(* Logix 5000 project; controller reports 1756-L63 rev 20.11; software revision 20.04; part 49 of 52 *)

        [172].log_data[23].time := 3600.0, [172].log_data[23].valid := 1, [172].log_data[24].time := 3600.0, [172].log_data[24].valid := 1, [172].log_data[25].time := 3600.0, [172].log_data[25].valid := 1, [172].log_data[26].time := 3600.0, [172].log_data[26].valid := 1, [172].log_data[27].time := 3600.0, [172].log_data[27].valid := 1, [172].log_data[28].time := 3600.0, [172].log_data[28].valid := 1, [172].log_data[29].min := 1.0, [172].log_data[29].max := 1.0, [172].log_data[29].total := 3600.0, [172].log_data[29].time := 3600.0, [172].log_data[29].valid := 1, [172].log_data[30].min := 1.0, [172].log_data[30].max := 1.0, [172].log_data[30].total := 3600.0, [172].log_data[30].time := 3600.0, [172].log_data[30].valid := 1, [172].log_data[31].max := 1.0, [172].log_data[31].total := 1629.7471, [172].log_data[31].time := 3600.0, [172].log_data[31].maxminute := 1, [172].log_data[31].valid := 1, [172].log_data[32].max := 1.0, [172].log_data[32].total := 1452.2471, [172].log_data[32].time := 3600.0, [172].log_data[32].maxminute := 11, [172].log_data[32].valid := 1, [172].log_data[33].time := 3600.0, [172].log_data[33].valid := 1, [172].log_data[34].time := 3600.0, [172].log_data[34].valid := 1, [172].log_data[35].max := 1.0, [172].log_data[35].total := 1440.5, [172].log_data[35].time := 3600.0, [172].log_data[35].minminute := 2, [172].log_data[35].valid := 1, [172].log_data[36].max := 1.0, [172].log_data[36].total := 1629.7471, [172].log_data[36].time := 3600.0, [172].log_data[36].maxminute := 4, [172].log_data[36].valid := 1, [172].log_data[37].max := 6.994973, [172].log_data[37].total := 3548.4736, [172].log_data[37].time := 3600.0, [172].log_data[37].maxminute := 52, [172].log_data[37].valid := 1, [172].log_data[38].time := 3600.0, [172].log_data[38].valid := 1, [172].log_data[39].min := 0.9945885, [172].log_data[39].max := 1.0214411, [172].log_data[39].total := 3605.796, [172].log_data[39].time := 3600.0, [172].log_data[39].minminute := 44, [172].log_data[39].maxminute := 58, [172].log_data[39].valid := 1,
        [172].log_data[40].min := 7.5503016, [172].log_data[40].max := 7.5794306, [172].log_data[40].total := 27251.781, [172].log_data[40].time := 3600.0, [172].log_data[40].minminute := 51, [172].log_data[40].maxminute := 15, [172].log_data[40].valid := 1, [172].log_data[41].min := 0.07907203, [172].log_data[41].max := 0.10674902, [172].log_data[41].total := 334.01642, [172].log_data[41].time := 3600.0, [172].log_data[41].minminute := 58, [172].log_data[41].valid := 1, [172].log_data[42].min := 2.293056, [172].log_data[42].max := 2.2978847, [172].log_data[42].total := 8264.451, [172].log_data[42].time := 3600.0, [172].log_data[42].minminute := 29, [172].log_data[42].maxminute := 2, [172].log_data[42].valid := 1, [172].log_data[43].min := -0.27999878, [172].log_data[43].max := -0.26000214, [172].log_data[43].total := -954.9988, [172].log_data[43].time := 3600.0, [172].log_data[43].valid := 1, [172].log_data[44].min := -0.30000305, [172].log_data[44].max := -0.27999878, [172].log_data[44].total := -1079.6469, [172].log_data[44].time := 3600.0, [172].log_data[44].maxminute := 4, [172].log_data[44].valid := 1, [172].log_data[45].time := 3600.0, [172].log_data[45].valid := 1, [172].log_data[46].time := 3600.0, [172].log_data[46].valid := 1, [172].log_data[47].time := 3600.0, [172].log_data[47].valid := 1, [172].log_data[48].min := 6.583802, [172].log_data[48].max := 6.9311595, [172].log_data[48].total := 24306.4, [172].log_data[48].time := 3600.0, [172].log_data[48].minminute := 5, [172].log_data[48].maxminute := 59, [172].log_data[48].valid := 1, [172].log_data[49].min := 6.690951, [172].log_data[49].max := 9.500274, [172].log_data[49].total := 31090.45, [172].log_data[49].time := 3600.0, [172].log_data[49].maxminute := 53, [172].log_data[49].valid := 1, [172].log_data[50].min := 2.067046, [172].log_data[50].max := 2.172219, [172].log_data[50].total := 7593.68, [172].log_data[50].time := 3600.0, [172].log_data[50].minminute := 51, [172].log_data[50].maxminute := 59, [172].log_data[50].valid := 1, [172].log_data[51].time := 3600.0, [172].log_data[51].valid := 1, [172].log_data[52].min := -3.0,
        [172].log_data[52].max := 0.11999512, [172].log_data[52].total := -7550.291, [172].log_data[52].time := 3600.0, [172].log_data[52].minminute := 43, [172].log_data[52].valid := 1, [172].log_data[53].min := -2.5, [172].log_data[53].max := 0.2599945, [172].log_data[53].total := -7057.6147, [172].log_data[53].time := 3600.0, [172].log_data[53].minminute := 14, [172].log_data[53].maxminute := 35, [172].log_data[53].valid := 1, [172].log_data[54].max := 0.56, [172].log_data[54].total := 1221.5302, [172].log_data[54].time := 3600.0, [172].log_data[54].maxminute := 1, [172].log_data[54].valid := 1, [172].log_data[55].max := 0.55799997, [172].log_data[55].total := 1217.0685, [172].log_data[55].time := 3600.0, [172].log_data[55].minminute := 2, [172].log_data[55].maxminute := 14, [172].log_data[55].valid := 1, [172].log_data[56].min := 0.16067745, [172].log_data[56].max := 0.16114853, [172].log_data[56].total := 579.2485, [172].log_data[56].time := 3600.0, [172].log_data[56].minminute := 9, [172].log_data[56].maxminute := 1, [172].log_data[56].valid := 1, [172].log_data[57].min := 0.34574097, [172].log_data[57].max := 0.3479787, [172].log_data[57].total := 1245.9099, [172].log_data[57].time := 3600.0, [172].log_data[57].minminute := 14, [172].log_data[57].maxminute := 1, [172].log_data[57].valid := 1, [172].log_data[58].time := 3600.0, [172].log_data[58].valid := 1, [172].log_data[59].time := 3600.0, [172].log_data[59].valid := 1, [172].log_data[60].valid := 1, [172].log_data[61].valid := 1, [172].log_data[62].valid := 1, [172].log_data[63].valid := 1, [172].log_data[64].valid := 1, [172].log_data[65].valid := 1, [172].log_data[66].valid := 1, [172].log_data[67].valid := 1, [172].log_data[68].valid := 1, [172].log_data[69].valid := 1, [172].log_data[70].valid := 1, [172].log_data[71].valid := 1, [172].log_data[72].valid := 1, [172].log_data[73].valid := 1, [172].log_data[74].valid := 1, [172].log_data[75].valid := 1, [172].log_data[76].valid := 1, [172].log_data[77].valid := 1, [172].log_data[78].valid := 1,
        [172].log_data[79].valid := 1, [172].log_data[80].valid := 1, [172].log_data[81].valid := 1, [172].log_data[82].valid := 1, [172].log_data[83].valid := 1, [172].log_data[84].valid := 1, [172].log_data[85].valid := 1, [172].log_data[86].valid := 1, [172].log_data[87].valid := 1, [172].log_data[88].valid := 1, [172].log_data[89].valid := 1, [172].log_data[90].valid := 1, [172].log_data[91].valid := 1, [172].log_data[92].valid := 1, [172].log_data[93].valid := 1, [172].log_data[94].valid := 1, [172].log_data[95].valid := 1, [172].log_data[96].valid := 1, [172].log_data[97].valid := 1, [172].log_data[98].valid := 1, [172].log_data[99].valid := 1, [172].log_data[100].valid := 1, [172].log_data[101].valid := 1, [172].log_data[102].valid := 1, [172].log_data[103].valid := 1, [172].log_data[104].valid := 1, [172].log_data[105].valid := 1, [172].log_data[106].valid := 1, [172].log_data[107].valid := 1, [172].log_data[108].valid := 1, [172].log_data[109].valid := 1, [172].log_data[110].valid := 1, [172].log_data[111].valid := 1, [172].log_data[112].valid := 1, [172].log_data[113].valid := 1, [172].log_data[114].valid := 1, [172].log_data[115].valid := 1, [172].log_data[116].valid := 1, [172].log_data[117].valid := 1, [172].log_data[118].valid := 1, [172].log_data[119].valid := 1, [172].log_data[120].valid := 1, [172].log_data[121].valid := 1, [172].log_data[122].valid := 1, [172].log_data[123].valid := 1, [172].log_data[124].valid := 1, [172].time.Year := 2023, [172].time.Month := 1, [172].time.Day := 11, [172].time.Hour := 23, [172].time.Minute := 59, [172].time.Second := 59, [173].log_data[0].min := 1.0, [173].log_data[0].max := 1.0, [173].log_data[0].total := 3600.0, [173].log_data[0].time := 3600.0, [173].log_data[0].valid := 1, [173].log_data[1].max := 1.0, [173].log_data[1].total := 26.251, [173].log_data[1].time := 3600.0,
        [173].log_data[1].valid := 1, [173].log_data[2].max := 1.0, [173].log_data[2].total := 26.251, [173].log_data[2].time := 3600.0, [173].log_data[2].valid := 1, [173].log_data[3].time := 3600.0, [173].log_data[3].valid := 1, [173].log_data[4].time := 3600.0, [173].log_data[4].valid := 1, [173].log_data[5].time := 3600.0, [173].log_data[5].valid := 1, [173].log_data[6].time := 3600.0, [173].log_data[6].valid := 1, [173].log_data[7].time := 3600.0, [173].log_data[7].valid := 1, [173].log_data[8].min := 1.0, [173].log_data[8].max := 1.0, [173].log_data[8].total := 3600.0, [173].log_data[8].time := 3600.0, [173].log_data[8].valid := 1, [173].log_data[9].min := 1.0, [173].log_data[9].max := 1.0, [173].log_data[9].total := 3600.0, [173].log_data[9].time := 3600.0, [173].log_data[9].valid := 1, [173].log_data[10].min := 1.0, [173].log_data[10].max := 1.0, [173].log_data[10].total := 3600.0, [173].log_data[10].time := 3600.0, [173].log_data[10].valid := 1, [173].log_data[11].time := 3600.0, [173].log_data[11].valid := 1, [173].log_data[12].min := 1.0, [173].log_data[12].max := 1.0, [173].log_data[12].total := 3600.0, [173].log_data[12].time := 3600.0, [173].log_data[12].valid := 1, [173].log_data[13].min := 1.0, [173].log_data[13].max := 1.0, [173].log_data[13].total := 3600.0, [173].log_data[13].time := 3600.0, [173].log_data[13].valid := 1, [173].log_data[14].time := 3600.0, [173].log_data[14].valid := 1, [173].log_data[15].time := 3600.0, [173].log_data[15].valid := 1, [173].log_data[16].time := 3600.0, [173].log_data[16].valid := 1, [173].log_data[17].min := 1.0, [173].log_data[17].max := 1.0, [173].log_data[17].total := 3600.0, [173].log_data[17].time := 3600.0, [173].log_data[17].valid := 1, [173].log_data[18].time := 3600.0, [173].log_data[18].valid := 1, [173].log_data[19].time := 3600.0, [173].log_data[19].valid := 1, [173].log_data[20].time := 3600.0, [173].log_data[20].valid := 1, [173].log_data[21].min := 1.0,
        [173].log_data[21].max := 1.0, [173].log_data[21].total := 3600.0, [173].log_data[21].time := 3600.0, [173].log_data[21].valid := 1, [173].log_data[22].time := 3600.0, [173].log_data[22].valid := 1, [173].log_data[23].time := 3600.0, [173].log_data[23].valid := 1, [173].log_data[24].time := 3600.0, [173].log_data[24].valid := 1, [173].log_data[25].time := 3600.0, [173].log_data[25].valid := 1, [173].log_data[26].time := 3600.0, [173].log_data[26].valid := 1, [173].log_data[27].time := 3600.0, [173].log_data[27].valid := 1, [173].log_data[28].time := 3600.0, [173].log_data[28].valid := 1, [173].log_data[29].min := 1.0, [173].log_data[29].max := 1.0, [173].log_data[29].total := 3600.0, [173].log_data[29].time := 3600.0, [173].log_data[29].valid := 1, [173].log_data[30].min := 1.0, [173].log_data[30].max := 1.0, [173].log_data[30].total := 3600.0, [173].log_data[30].time := 3600.0, [173].log_data[30].valid := 1, [173].log_data[31].max := 1.0, [173].log_data[31].total := 1629.7471, [173].log_data[31].time := 3600.0, [173].log_data[31].maxminute := 4, [173].log_data[31].valid := 1, [173].log_data[32].max := 1.0, [173].log_data[32].total := 1440.7471, [173].log_data[32].time := 3600.0, [173].log_data[32].minminute := 2, [173].log_data[32].valid := 1, [173].log_data[33].time := 3600.0, [173].log_data[33].valid := 1, [173].log_data[34].time := 3600.0, [173].log_data[34].valid := 1, [173].log_data[35].max := 1.0, [173].log_data[35].total := 1443.498, [173].log_data[35].time := 3600.0, [173].log_data[35].minminute := 5, [173].log_data[35].valid := 1, [173].log_data[36].max := 1.0, [173].log_data[36].total := 1629.7471, [173].log_data[36].time := 3600.0, [173].log_data[36].maxminute := 7, [173].log_data[36].valid := 1, [173].log_data[37].time := 3600.0, [173].log_data[37].valid := 1, [173].log_data[38].time := 3600.0, [173].log_data[38].valid := 1, [173].log_data[39].min := 0.995884, [173].log_data[39].max := 1.0066015, [173].log_data[39].total := 3607.993, [173].log_data[39].time := 3600.0,
        [173].log_data[39].minminute := 43, [173].log_data[39].maxminute := 56, [173].log_data[39].valid := 1, [173].log_data[40].min := 7.553049, [173].log_data[40].max := 7.5832787, [173].log_data[40].total := 27256.387, [173].log_data[40].time := 3600.0, [173].log_data[40].minminute := 13, [173].log_data[40].maxminute := 18, [173].log_data[40].valid := 1, [173].log_data[41].min := 0.08005347, [173].log_data[41].max := 0.13226709, [173].log_data[41].total := 406.6626, [173].log_data[41].time := 3600.0, [173].log_data[41].maxminute := 31, [173].log_data[41].valid := 1, [173].log_data[42].min := 2.293056, [173].log_data[42].max := 2.2978847, [173].log_data[42].total := 8264.515, [173].log_data[42].time := 3600.0, [173].log_data[42].minminute := 12, [173].log_data[42].maxminute := 45, [173].log_data[42].valid := 1, [173].log_data[43].min := -0.27999878, [173].log_data[43].max := -0.26000214, [173].log_data[43].total := -953.048, [173].log_data[43].time := 3600.0, [173].log_data[43].valid := 1, [173].log_data[44].min := -0.30000305, [173].log_data[44].max := -0.27999878, [173].log_data[44].total := -1078.877, [173].log_data[44].time := 3600.0, [173].log_data[44].maxminute := 4, [173].log_data[44].valid := 1, [173].log_data[45].time := 3600.0, [173].log_data[45].valid := 1, [173].log_data[46].time := 3600.0, [173].log_data[46].valid := 1, [173].log_data[47].time := 3600.0, [173].log_data[47].valid := 1, [173].log_data[48].min := 6.5983667, [173].log_data[48].max := 6.903678, [173].log_data[48].total := 24199.447, [173].log_data[48].time := 3600.0, [173].log_data[48].minminute := 23, [173].log_data[48].valid := 1, [173].log_data[49].min := 6.840722, [173].log_data[49].max := 9.401342, [173].log_data[49].total := 29274.203, [173].log_data[49].time := 3600.0, [173].log_data[49].minminute := 20, [173].log_data[49].maxminute := 59, [173].log_data[49].valid := 1, [173].log_data[50].min := 2.0936632, [173].log_data[50].max := 2.1728077, [173].log_data[50].total := 7691.275, [173].log_data[50].time := 3600.0, [173].log_data[50].minminute := 59, [173].log_data[50].valid := 1, [173].log_data[51].time := 3600.0,
        [173].log_data[51].valid := 1, [173].log_data[52].min := -2.959999, [173].log_data[52].max := 0.11999512, [173].log_data[52].total := -7556.767, [173].log_data[52].time := 3600.0, [173].log_data[52].minminute := 25, [173].log_data[52].maxminute := 3, [173].log_data[52].valid := 1, [173].log_data[53].min := -2.5, [173].log_data[53].max := 0.2400055, [173].log_data[53].total := -7110.352, [173].log_data[53].time := 3600.0, [173].log_data[53].minminute := 42, [173].log_data[53].maxminute := 17, [173].log_data[53].valid := 1, [173].log_data[54].max := 0.528, [173].log_data[54].total := 1217.4906, [173].log_data[54].time := 3600.0, [173].log_data[54].minminute := 2, [173].log_data[54].maxminute := 25, [173].log_data[54].valid := 1, [173].log_data[55].max := 0.525, [173].log_data[55].total := 1220.6111, [173].log_data[55].time := 3600.0, [173].log_data[55].minminute := 5, [173].log_data[55].maxminute := 39, [173].log_data[55].valid := 1, [173].log_data[56].min := 0.1607167, [173].log_data[56].max := 0.16110928, [173].log_data[56].total := 579.1586, [173].log_data[56].time := 3600.0, [173].log_data[56].minminute := 47, [173].log_data[56].maxminute := 6, [173].log_data[56].valid := 1, [173].log_data[57].min := 0.3444062, [173].log_data[57].max := 0.34609428, [173].log_data[57].total := 1242.74, [173].log_data[57].time := 3600.0, [173].log_data[57].minminute := 35, [173].log_data[57].maxminute := 1, [173].log_data[57].valid := 1, [173].log_data[58].time := 3600.0, [173].log_data[58].valid := 1, [173].log_data[59].time := 3600.0, [173].log_data[59].valid := 1, [173].log_data[60].valid := 1, [173].log_data[61].valid := 1, [173].log_data[62].valid := 1, [173].log_data[63].valid := 1, [173].log_data[64].valid := 1, [173].log_data[65].valid := 1, [173].log_data[66].valid := 1, [173].log_data[67].valid := 1, [173].log_data[68].valid := 1, [173].log_data[69].valid := 1, [173].log_data[70].valid := 1, [173].log_data[71].valid := 1, [173].log_data[72].valid := 1, [173].log_data[73].valid := 1, [173].log_data[74].valid := 1,
        [173].log_data[75].valid := 1, [173].log_data[76].valid := 1, [173].log_data[77].valid := 1, [173].log_data[78].valid := 1, [173].log_data[79].valid := 1, [173].log_data[80].valid := 1, [173].log_data[81].valid := 1, [173].log_data[82].valid := 1, [173].log_data[83].valid := 1, [173].log_data[84].valid := 1, [173].log_data[85].valid := 1, [173].log_data[86].valid := 1, [173].log_data[87].valid := 1, [173].log_data[88].valid := 1, [173].log_data[89].valid := 1, [173].log_data[90].valid := 1, [173].log_data[91].valid := 1, [173].log_data[92].valid := 1, [173].log_data[93].valid := 1, [173].log_data[94].valid := 1, [173].log_data[95].valid := 1, [173].log_data[96].valid := 1, [173].log_data[97].valid := 1, [173].log_data[98].valid := 1, [173].log_data[99].valid := 1, [173].log_data[100].valid := 1, [173].log_data[101].valid := 1, [173].log_data[102].valid := 1, [173].log_data[103].valid := 1, [173].log_data[104].valid := 1, [173].log_data[105].valid := 1, [173].log_data[106].valid := 1, [173].log_data[107].valid := 1, [173].log_data[108].valid := 1, [173].log_data[109].valid := 1, [173].log_data[110].valid := 1, [173].log_data[111].valid := 1, [173].log_data[112].valid := 1, [173].log_data[113].valid := 1, [173].log_data[114].valid := 1, [173].log_data[115].valid := 1, [173].log_data[116].valid := 1, [173].log_data[117].valid := 1, [173].log_data[118].valid := 1, [173].log_data[119].valid := 1, [173].log_data[120].valid := 1, [173].log_data[121].valid := 1, [173].log_data[122].valid := 1, [173].log_data[123].valid := 1, [173].log_data[124].valid := 1, [173].time.Year := 2023, [173].time.Month := 1, [173].time.Day := 12, [173].time.Minute := 59, [173].time.Second := 59, [174].log_data[0].min := 1.0, [174].log_data[0].max := 1.0, [174].log_data[0].total := 3599.5, [174].log_data[0].time := 3599.5, [174].log_data[0].valid := 1,
        [174].log_data[1].time := 3599.5, [174].log_data[1].valid := 1, [174].log_data[2].time := 3599.5, [174].log_data[2].valid := 1, [174].log_data[3].time := 3599.5, [174].log_data[3].valid := 1, [174].log_data[4].time := 3599.5, [174].log_data[4].valid := 1, [174].log_data[5].time := 3599.5, [174].log_data[5].valid := 1, [174].log_data[6].time := 3599.5, [174].log_data[6].valid := 1, [174].log_data[7].time := 3599.5, [174].log_data[7].valid := 1, [174].log_data[8].min := 1.0, [174].log_data[8].max := 1.0, [174].log_data[8].total := 3599.5, [174].log_data[8].time := 3599.5, [174].log_data[8].valid := 1, [174].log_data[9].min := 1.0, [174].log_data[9].max := 1.0, [174].log_data[9].total := 3599.5, [174].log_data[9].time := 3599.5, [174].log_data[9].valid := 1, [174].log_data[10].min := 1.0, [174].log_data[10].max := 1.0, [174].log_data[10].total := 3599.5, [174].log_data[10].time := 3599.5, [174].log_data[10].valid := 1, [174].log_data[11].time := 3599.5, [174].log_data[11].valid := 1, [174].log_data[12].min := 1.0, [174].log_data[12].max := 1.0, [174].log_data[12].total := 3599.5, [174].log_data[12].time := 3599.5, [174].log_data[12].valid := 1, [174].log_data[13].min := 1.0, [174].log_data[13].max := 1.0, [174].log_data[13].total := 3599.5, [174].log_data[13].time := 3599.5, [174].log_data[13].valid := 1, [174].log_data[14].time := 3599.5, [174].log_data[14].valid := 1, [174].log_data[15].time := 3599.5, [174].log_data[15].valid := 1, [174].log_data[16].time := 3599.5, [174].log_data[16].valid := 1, [174].log_data[17].min := 1.0, [174].log_data[17].max := 1.0, [174].log_data[17].total := 3599.5, [174].log_data[17].time := 3599.5, [174].log_data[17].valid := 1, [174].log_data[18].time := 3599.5, [174].log_data[18].valid := 1, [174].log_data[19].time := 3599.5, [174].log_data[19].valid := 1, [174].log_data[20].time := 3599.5, [174].log_data[20].valid := 1, [174].log_data[21].min := 1.0, [174].log_data[21].max := 1.0,
        [174].log_data[21].total := 3599.5, [174].log_data[21].time := 3599.5, [174].log_data[21].valid := 1, [174].log_data[22].time := 3599.5, [174].log_data[22].valid := 1, [174].log_data[23].time := 3599.5, [174].log_data[23].valid := 1, [174].log_data[24].time := 3599.5, [174].log_data[24].valid := 1, [174].log_data[25].time := 3599.5, [174].log_data[25].valid := 1, [174].log_data[26].time := 3599.5, [174].log_data[26].valid := 1, [174].log_data[27].time := 3599.5, [174].log_data[27].valid := 1, [174].log_data[28].time := 3599.5, [174].log_data[28].valid := 1, [174].log_data[29].min := 1.0, [174].log_data[29].max := 1.0, [174].log_data[29].total := 3599.5, [174].log_data[29].time := 3599.5, [174].log_data[29].valid := 1, [174].log_data[30].min := 1.0, [174].log_data[30].max := 1.0, [174].log_data[30].total := 3599.5, [174].log_data[30].time := 3599.5, [174].log_data[30].valid := 1, [174].log_data[31].max := 1.0, [174].log_data[31].total := 1629.7471, [174].log_data[31].time := 3599.5, [174].log_data[31].maxminute := 7, [174].log_data[31].valid := 1, [174].log_data[32].max := 1.0, [174].log_data[32].total := 1452.998, [174].log_data[32].time := 3599.5, [174].log_data[32].minminute := 6, [174].log_data[32].valid := 1, [174].log_data[33].time := 3599.5, [174].log_data[33].valid := 1, [174].log_data[34].time := 3599.5, [174].log_data[34].valid := 1, [174].log_data[35].max := 1.0, [174].log_data[35].total := 1629.7471, [174].log_data[35].time := 3599.5, [174].log_data[35].valid := 1, [174].log_data[36].max := 1.0, [174].log_data[36].total := 1525.7471, [174].log_data[36].time := 3599.5, [174].log_data[36].maxminute := 10, [174].log_data[36].valid := 1, [174].log_data[37].time := 3599.5, [174].log_data[37].valid := 1, [174].log_data[38].time := 3599.5, [174].log_data[38].valid := 1, [174].log_data[39].min := 0.9956484, [174].log_data[39].max := 1.0071905, [174].log_data[39].total := 3608.351, [174].log_data[39].time := 3599.5, [174].log_data[39].minminute := 10, [174].log_data[39].maxminute := 23,
        [174].log_data[39].valid := 1, [174].log_data[40].min := 7.5390344, [174].log_data[40].max := 7.592072, [174].log_data[40].total := 27246.436, [174].log_data[40].time := 3599.5, [174].log_data[40].minminute := 9, [174].log_data[40].maxminute := 18, [174].log_data[40].valid := 1, [174].log_data[41].min := 0.08613843, [174].log_data[41].max := 0.14345556, [174].log_data[41].total := 424.99884, [174].log_data[41].time := 3599.5, [174].log_data[41].minminute := 29, [174].log_data[41].maxminute := 56, [174].log_data[41].valid := 1, [174].log_data[42].min := 2.293056, [174].log_data[42].max := 2.2980025, [174].log_data[42].total := 8263.423, [174].log_data[42].time := 3599.5, [174].log_data[42].minminute := 20, [174].log_data[42].maxminute := 44, [174].log_data[42].valid := 1, [174].log_data[43].min := -0.27999878, [174].log_data[43].max := -0.26000214, [174].log_data[43].total := -944.1006, [174].log_data[43].time := 3599.5, [174].log_data[43].valid := 1, [174].log_data[44].min := -0.30000305, [174].log_data[44].max := -0.27999878, [174].log_data[44].total := -1079.4894, [174].log_data[44].time := 3599.5, [174].log_data[44].maxminute := 6, [174].log_data[44].valid := 1, [174].log_data[45].time := 3599.5, [174].log_data[45].valid := 1, [174].log_data[46].time := 3599.5, [174].log_data[46].valid := 1, [174].log_data[47].time := 3599.5, [174].log_data[47].valid := 1, [174].log_data[48].min := 6.753908, [174].log_data[48].max := 6.762702, [174].log_data[48].total := 24325.047, [174].log_data[48].time := 3599.5, [174].log_data[48].minminute := 58, [174].log_data[48].maxminute := 2, [174].log_data[48].valid := 1, [174].log_data[49].min := 9.398202, [174].log_data[49].max := 9.565442, [174].log_data[49].total := 34182.1, [174].log_data[49].time := 3599.5, [174].log_data[49].maxminute := 52, [174].log_data[49].valid := 1, [174].log_data[50].min := 2.006392, [174].log_data[50].max := 2.1013186, [174].log_data[50].total := 7397.241, [174].log_data[50].time := 3599.5, [174].log_data[50].minminute := 59, [174].log_data[50].valid := 1, [174].log_data[51].time := 3599.5, [174].log_data[51].valid := 1,
        [174].log_data[52].min := -3.0800018, [174].log_data[52].max := 0.11999512, [174].log_data[52].total := -7629.0737, [174].log_data[52].time := 3599.5, [174].log_data[52].minminute := 7, [174].log_data[52].maxminute := 6, [174].log_data[52].valid := 1, [174].log_data[53].min := -2.5200043, [174].log_data[53].max := 0.19999695, [174].log_data[53].total := -7349.1704, [174].log_data[53].time := 3599.5, [174].log_data[53].minminute := 57, [174].log_data[53].valid := 1, [174].log_data[54].max := 0.559, [174].log_data[54].total := 1224.2659, [174].log_data[54].time := 3599.5, [174].log_data[54].minminute := 6, [174].log_data[54].maxminute := 7, [174].log_data[54].valid := 1, [174].log_data[55].max := 0.528, [174].log_data[55].total := 1250.9253, [174].log_data[55].time := 3599.5, [174].log_data[55].maxminute := 31, [174].log_data[55].valid := 1, [174].log_data[56].min := 0.16067745, [174].log_data[56].max := 0.16110928, [174].log_data[56].total := 578.99304, [174].log_data[56].time := 3599.5, [174].log_data[56].minminute := 34, [174].log_data[56].maxminute := 6, [174].log_data[56].valid := 1, [174].log_data[57].min := 0.3444062, [174].log_data[57].max := 0.34483802, [174].log_data[57].total := 1240.3518, [174].log_data[57].time := 3599.5, [174].log_data[57].minminute := 38, [174].log_data[57].maxminute := 11, [174].log_data[57].valid := 1, [174].log_data[58].time := 3599.5, [174].log_data[58].valid := 1, [174].log_data[59].time := 3599.5, [174].log_data[59].valid := 1, [174].log_data[60].valid := 1, [174].log_data[61].valid := 1, [174].log_data[62].valid := 1, [174].log_data[63].valid := 1, [174].log_data[64].valid := 1, [174].log_data[65].valid := 1, [174].log_data[66].valid := 1, [174].log_data[67].valid := 1, [174].log_data[68].valid := 1, [174].log_data[69].valid := 1, [174].log_data[70].valid := 1, [174].log_data[71].valid := 1, [174].log_data[72].valid := 1, [174].log_data[73].valid := 1, [174].log_data[74].valid := 1, [174].log_data[75].valid := 1, [174].log_data[76].valid := 1, [174].log_data[77].valid := 1,
        [174].log_data[78].valid := 1, [174].log_data[79].valid := 1, [174].log_data[80].valid := 1, [174].log_data[81].valid := 1, [174].log_data[82].valid := 1, [174].log_data[83].valid := 1, [174].log_data[84].valid := 1, [174].log_data[85].valid := 1, [174].log_data[86].valid := 1, [174].log_data[87].valid := 1, [174].log_data[88].valid := 1, [174].log_data[89].valid := 1, [174].log_data[90].valid := 1, [174].log_data[91].valid := 1, [174].log_data[92].valid := 1, [174].log_data[93].valid := 1, [174].log_data[94].valid := 1, [174].log_data[95].valid := 1, [174].log_data[96].valid := 1, [174].log_data[97].valid := 1, [174].log_data[98].valid := 1, [174].log_data[99].valid := 1, [174].log_data[100].valid := 1, [174].log_data[101].valid := 1, [174].log_data[102].valid := 1, [174].log_data[103].valid := 1, [174].log_data[104].valid := 1, [174].log_data[105].valid := 1, [174].log_data[106].valid := 1, [174].log_data[107].valid := 1, [174].log_data[108].valid := 1, [174].log_data[109].valid := 1, [174].log_data[110].valid := 1, [174].log_data[111].valid := 1, [174].log_data[112].valid := 1, [174].log_data[113].valid := 1, [174].log_data[114].valid := 1, [174].log_data[115].valid := 1, [174].log_data[116].valid := 1, [174].log_data[117].valid := 1, [174].log_data[118].valid := 1, [174].log_data[119].valid := 1, [174].log_data[120].valid := 1, [174].log_data[121].valid := 1, [174].log_data[122].valid := 1, [174].log_data[123].valid := 1, [174].log_data[124].valid := 1, [174].time.Year := 2023, [174].time.Month := 1, [174].time.Day := 12, [174].time.Hour := 1, [174].time.Minute := 59, [174].time.Second := 59, [175].log_data[0].min := 1.0, [175].log_data[0].max := 1.0, [175].log_data[0].total := 3600.0, [175].log_data[0].time := 3600.0, [175].log_data[0].valid := 1, [175].log_data[1].max := 1.0, [175].log_data[1].total := 524.0,
        [175].log_data[1].time := 3600.0, [175].log_data[1].maxminute := 21, [175].log_data[1].valid := 1, [175].log_data[2].max := 1.0, [175].log_data[2].total := 520.5, [175].log_data[2].time := 3600.0, [175].log_data[2].maxminute := 21, [175].log_data[2].valid := 1, [175].log_data[3].time := 3600.0, [175].log_data[3].valid := 1, [175].log_data[4].time := 3600.0, [175].log_data[4].valid := 1, [175].log_data[5].max := 1.0, [175].log_data[5].total := 237.0, [175].log_data[5].time := 3600.0, [175].log_data[5].maxminute := 23, [175].log_data[5].valid := 1, [175].log_data[6].time := 3600.0, [175].log_data[6].valid := 1, [175].log_data[7].time := 3600.0, [175].log_data[7].valid := 1, [175].log_data[8].max := 1.0, [175].log_data[8].total := 2444.5, [175].log_data[8].time := 3600.0, [175].log_data[8].minminute := 5, [175].log_data[8].valid := 1, [175].log_data[9].max := 1.0, [175].log_data[9].total := 2441.0, [175].log_data[9].time := 3600.0, [175].log_data[9].minminute := 5, [175].log_data[9].valid := 1, [175].log_data[10].min := 1.0, [175].log_data[10].max := 1.0, [175].log_data[10].total := 3600.0, [175].log_data[10].time := 3600.0, [175].log_data[10].valid := 1, [175].log_data[11].time := 3600.0, [175].log_data[11].valid := 1, [175].log_data[12].min := 1.0, [175].log_data[12].max := 1.0, [175].log_data[12].total := 3600.0, [175].log_data[12].time := 3600.0, [175].log_data[12].valid := 1, [175].log_data[13].min := 1.0, [175].log_data[13].max := 1.0, [175].log_data[13].total := 3600.0, [175].log_data[13].time := 3600.0, [175].log_data[13].valid := 1, [175].log_data[14].time := 3600.0, [175].log_data[14].valid := 1, [175].log_data[15].time := 3600.0, [175].log_data[15].valid := 1, [175].log_data[16].time := 3600.0, [175].log_data[16].valid := 1, [175].log_data[17].min := 1.0, [175].log_data[17].max := 1.0, [175].log_data[17].total := 3600.0, [175].log_data[17].time := 3600.0, [175].log_data[17].valid := 1, [175].log_data[18].time := 3600.0,
        [175].log_data[18].valid := 1, [175].log_data[19].time := 3600.0, [175].log_data[19].valid := 1, [175].log_data[20].time := 3600.0, [175].log_data[20].valid := 1, [175].log_data[21].min := 1.0, [175].log_data[21].max := 1.0, [175].log_data[21].total := 3600.0, [175].log_data[21].time := 3600.0, [175].log_data[21].valid := 1, [175].log_data[22].time := 3600.0, [175].log_data[22].valid := 1, [175].log_data[23].time := 3600.0, [175].log_data[23].valid := 1, [175].log_data[24].time := 3600.0, [175].log_data[24].valid := 1, [175].log_data[25].time := 3600.0, [175].log_data[25].valid := 1, [175].log_data[26].time := 3600.0, [175].log_data[26].valid := 1, [175].log_data[27].time := 3600.0, [175].log_data[27].valid := 1, [175].log_data[28].time := 3600.0, [175].log_data[28].valid := 1, [175].log_data[29].min := 1.0, [175].log_data[29].max := 1.0, [175].log_data[29].total := 3600.0, [175].log_data[29].time := 3600.0, [175].log_data[29].valid := 1, [175].log_data[30].min := 1.0, [175].log_data[30].max := 1.0, [175].log_data[30].total := 3600.0, [175].log_data[30].time := 3600.0, [175].log_data[30].valid := 1, [175].log_data[31].max := 1.0, [175].log_data[31].total := 736.998, [175].log_data[31].time := 3600.0, [175].log_data[31].maxminute := 25, [175].log_data[31].valid := 1, [175].log_data[32].max := 1.0, [175].log_data[32].total := 1426.998, [175].log_data[32].time := 3600.0, [175].log_data[32].valid := 1, [175].log_data[33].time := 3600.0, [175].log_data[33].valid := 1, [175].log_data[34].time := 3600.0, [175].log_data[34].valid := 1, [175].log_data[35].max := 1.0, [175].log_data[35].total := 1064.247, [175].log_data[35].time := 3600.0, [175].log_data[35].maxminute := 3, [175].log_data[35].valid := 1, [175].log_data[36].max := 1.0, [175].log_data[36].total := 1020.498, [175].log_data[36].time := 3600.0, [175].log_data[36].minminute := 1, [175].log_data[36].valid := 1, [175].log_data[37].max := 7.558722, [175].log_data[37].total := 3407.4478, [175].log_data[37].time := 3600.0,
        [175].log_data[37].maxminute := 21, [175].log_data[37].valid := 1, [175].log_data[38].time := 3600.0, [175].log_data[38].valid := 1, [175].log_data[39].min := 0.9945885, [175].log_data[39].max := 1.02097, [175].log_data[39].total := 3608.6638, [175].log_data[39].time := 3600.0, [175].log_data[39].minminute := 51, [175].log_data[39].maxminute := 23, [175].log_data[39].valid := 1, [175].log_data[40].min := 7.5379353, [175].log_data[40].max := 7.5794306, [175].log_data[40].total := 27251.215, [175].log_data[40].time := 3600.0, [175].log_data[40].minminute := 14, [175].log_data[40].maxminute := 16, [175].log_data[40].valid := 1, [175].log_data[41].min := 0.0963457, [175].log_data[41].max := 0.14031494, [175].log_data[41].total := 379.17615, [175].log_data[41].time := 3600.0, [175].log_data[41].minminute := 52, [175].log_data[41].valid := 1, [175].log_data[42].min := 2.2929382, [175].log_data[42].max := 2.2978847, [175].log_data[42].total := 8264.402, [175].log_data[42].time := 3600.0, [175].log_data[42].minminute := 46, [175].log_data[42].maxminute := 4, [175].log_data[42].valid := 1, [175].log_data[43].min := -0.27999878, [175].log_data[43].max := -0.26000214, [175].log_data[43].total := -943.9623, [175].log_data[43].time := 3600.0, [175].log_data[43].valid := 1, [175].log_data[44].min := -0.30000305, [175].log_data[44].max := -0.27999878, [175].log_data[44].total := -1079.5896, [175].log_data[44].time := 3600.0, [175].log_data[44].valid := 1, [175].log_data[45].time := 3600.0, [175].log_data[45].valid := 1, [175].log_data[46].time := 3600.0, [175].log_data[46].valid := 1, [175].log_data[47].time := 3600.0, [175].log_data[47].valid := 1, [175].log_data[48].min := 6.5810537, [175].log_data[48].max := 6.969357, [175].log_data[48].total := 24223.447, [175].log_data[48].time := 3600.0, [175].log_data[48].minminute := 53, [175].log_data[48].maxminute := 26, [175].log_data[48].valid := 1, [175].log_data[49].min := 6.7979293, [175].log_data[49].max := 9.501255, [175].log_data[49].total := 30011.445, [175].log_data[49].time := 3600.0, [175].log_data[49].minminute := 49, [175].log_data[49].valid := 1,
        [175].log_data[50].min := 1.9999144, [175].log_data[50].max := 2.1501951, [175].log_data[50].total := 7513.3774, [175].log_data[50].time := 3600.0, [175].log_data[50].minminute := 5, [175].log_data[50].maxminute := 25, [175].log_data[50].valid := 1, [175].log_data[51].time := 3600.0, [175].log_data[51].valid := 1, [175].log_data[52].min := -4.1800003, [175].log_data[52].max := 0.11999512, [175].log_data[52].total := -6929.6797, [175].log_data[52].time := 3600.0, [175].log_data[52].minminute := 25, [175].log_data[52].valid := 1, [175].log_data[53].min := -3.9199982, [175].log_data[53].max := 0.19999695, [175].log_data[53].total := -6288.31, [175].log_data[53].time := 3600.0, [175].log_data[53].minminute := 25, [175].log_data[53].maxminute := 32, [175].log_data[53].valid := 1, [175].log_data[54].max := 0.51, [175].log_data[54].total := 855.8069, [175].log_data[54].time := 3600.0, [175].log_data[54].valid := 1, [175].log_data[55].max := 0.514, [175].log_data[55].total := 824.69495, [175].log_data[55].time := 3600.0, [175].log_data[55].minminute := 1, [175].log_data[55].maxminute := 33, [175].log_data[55].valid := 1, [175].log_data[56].min := 0.16063818, [175].log_data[56].max := 0.16107002, [175].log_data[56].total := 578.963, [175].log_data[56].time := 3600.0, [175].log_data[56].minminute := 56, [175].log_data[56].maxminute := 6, [175].log_data[56].valid := 1, [175].log_data[57].min := 0.3431499, [175].log_data[57].max := 0.34483802, [175].log_data[57].total := 1240.1224, [175].log_data[57].time := 3600.0, [175].log_data[57].minminute := 59, [175].log_data[57].maxminute := 43, [175].log_data[57].valid := 1, [175].log_data[58].time := 3600.0, [175].log_data[58].valid := 1, [175].log_data[59].time := 3600.0, [175].log_data[59].valid := 1, [175].log_data[60].valid := 1, [175].log_data[61].valid := 1, [175].log_data[62].valid := 1, [175].log_data[63].valid := 1, [175].log_data[64].valid := 1, [175].log_data[65].valid := 1, [175].log_data[66].valid := 1, [175].log_data[67].valid := 1, [175].log_data[68].valid := 1, [175].log_data[69].valid := 1,
        [175].log_data[70].valid := 1, [175].log_data[71].valid := 1, [175].log_data[72].valid := 1, [175].log_data[73].valid := 1, [175].log_data[74].valid := 1, [175].log_data[75].valid := 1, [175].log_data[76].valid := 1, [175].log_data[77].valid := 1, [175].log_data[78].valid := 1, [175].log_data[79].valid := 1, [175].log_data[80].valid := 1, [175].log_data[81].valid := 1, [175].log_data[82].valid := 1, [175].log_data[83].valid := 1, [175].log_data[84].valid := 1, [175].log_data[85].valid := 1, [175].log_data[86].valid := 1, [175].log_data[87].valid := 1, [175].log_data[88].valid := 1, [175].log_data[89].valid := 1, [175].log_data[90].valid := 1, [175].log_data[91].valid := 1, [175].log_data[92].valid := 1, [175].log_data[93].valid := 1, [175].log_data[94].valid := 1, [175].log_data[95].valid := 1, [175].log_data[96].valid := 1, [175].log_data[97].valid := 1, [175].log_data[98].valid := 1, [175].log_data[99].valid := 1, [175].log_data[100].valid := 1, [175].log_data[101].valid := 1, [175].log_data[102].valid := 1, [175].log_data[103].valid := 1, [175].log_data[104].valid := 1, [175].log_data[105].valid := 1, [175].log_data[106].valid := 1, [175].log_data[107].valid := 1, [175].log_data[108].valid := 1, [175].log_data[109].valid := 1, [175].log_data[110].valid := 1, [175].log_data[111].valid := 1, [175].log_data[112].valid := 1, [175].log_data[113].valid := 1, [175].log_data[114].valid := 1, [175].log_data[115].valid := 1, [175].log_data[116].valid := 1, [175].log_data[117].valid := 1, [175].log_data[118].valid := 1, [175].log_data[119].valid := 1, [175].log_data[120].valid := 1, [175].log_data[121].valid := 1, [175].log_data[122].valid := 1, [175].log_data[123].valid := 1, [175].log_data[124].valid := 1, [175].time.Year := 2023, [175].time.Month := 1, [175].time.Day := 12, [175].time.Hour := 2, [175].time.Minute := 59,
        [175].time.Second := 59, [176].log_data[0].min := 1.0, [176].log_data[0].max := 1.0, [176].log_data[0].total := 3600.0, [176].log_data[0].time := 3600.0, [176].log_data[0].valid := 1, [176].log_data[1].time := 3600.0, [176].log_data[1].valid := 1, [176].log_data[2].time := 3600.0, [176].log_data[2].valid := 1, [176].log_data[3].time := 3600.0, [176].log_data[3].valid := 1, [176].log_data[4].time := 3600.0, [176].log_data[4].valid := 1, [176].log_data[5].time := 3600.0, [176].log_data[5].valid := 1, [176].log_data[6].time := 3600.0, [176].log_data[6].valid := 1, [176].log_data[7].time := 3600.0, [176].log_data[7].valid := 1, [176].log_data[8].max := 1.0, [176].log_data[8].total := 2797.251, [176].log_data[8].time := 3600.0, [176].log_data[8].minminute := 46, [176].log_data[8].valid := 1, [176].log_data[9].max := 1.0, [176].log_data[9].total := 2797.251, [176].log_data[9].time := 3600.0, [176].log_data[9].minminute := 46, [176].log_data[9].valid := 1, [176].log_data[10].min := 1.0, [176].log_data[10].max := 1.0, [176].log_data[10].total := 3600.0, [176].log_data[10].time := 3600.0, [176].log_data[10].valid := 1, [176].log_data[11].time := 3600.0, [176].log_data[11].valid := 1, [176].log_data[12].min := 1.0, [176].log_data[12].max := 1.0, [176].log_data[12].total := 3600.0, [176].log_data[12].time := 3600.0, [176].log_data[12].valid := 1, [176].log_data[13].min := 1.0, [176].log_data[13].max := 1.0, [176].log_data[13].total := 3600.0, [176].log_data[13].time := 3600.0, [176].log_data[13].valid := 1, [176].log_data[14].time := 3600.0, [176].log_data[14].valid := 1, [176].log_data[15].time := 3600.0, [176].log_data[15].valid := 1, [176].log_data[16].time := 3600.0, [176].log_data[16].valid := 1, [176].log_data[17].min := 1.0, [176].log_data[17].max := 1.0, [176].log_data[17].total := 3600.0, [176].log_data[17].time := 3600.0, [176].log_data[17].valid := 1, [176].log_data[18].time := 3600.0, [176].log_data[18].valid := 1,
        [176].log_data[19].time := 3600.0, [176].log_data[19].valid := 1, [176].log_data[20].time := 3600.0, [176].log_data[20].valid := 1, [176].log_data[21].min := 1.0, [176].log_data[21].max := 1.0, [176].log_data[21].total := 3600.0, [176].log_data[21].time := 3600.0, [176].log_data[21].valid := 1, [176].log_data[22].time := 3600.0, [176].log_data[22].valid := 1, [176].log_data[23].time := 3600.0, [176].log_data[23].valid := 1, [176].log_data[24].time := 3600.0, [176].log_data[24].valid := 1, [176].log_data[25].time := 3600.0, [176].log_data[25].valid := 1, [176].log_data[26].time := 3600.0, [176].log_data[26].valid := 1, [176].log_data[27].time := 3600.0, [176].log_data[27].valid := 1, [176].log_data[28].time := 3600.0, [176].log_data[28].valid := 1, [176].log_data[29].min := 1.0, [176].log_data[29].max := 1.0, [176].log_data[29].total := 3600.0, [176].log_data[29].time := 3600.0, [176].log_data[29].valid := 1, [176].log_data[30].min := 1.0, [176].log_data[30].max := 1.0, [176].log_data[30].total := 3600.0, [176].log_data[30].time := 3600.0, [176].log_data[30].valid := 1, [176].log_data[31].max := 1.0, [176].log_data[31].total := 1263.749, [176].log_data[31].time := 3600.0, [176].log_data[31].maxminute := 1, [176].log_data[31].valid := 1, [176].log_data[32].max := 1.0, [176].log_data[32].total := 1095.749, [176].log_data[32].time := 3600.0, [176].log_data[32].valid := 1, [176].log_data[33].time := 3600.0, [176].log_data[33].valid := 1, [176].log_data[34].time := 3600.0, [176].log_data[34].valid := 1, [176].log_data[35].max := 1.0, [176].log_data[35].total := 1278.498, [176].log_data[35].time := 3600.0, [176].log_data[35].minminute := 3, [176].log_data[35].valid := 1, [176].log_data[36].max := 1.0, [176].log_data[36].total := 1086.498, [176].log_data[36].time := 3600.0, [176].log_data[36].maxminute := 4, [176].log_data[36].valid := 1, [176].log_data[37].time := 3600.0, [176].log_data[37].valid := 1, [176].log_data[38].time := 3600.0, [176].log_data[38].valid := 1,
        [176].log_data[39].min := 0.9941174, [176].log_data[39].max := 1.0041281, [176].log_data[39].total := 3599.7744, [176].log_data[39].time := 3600.0, [176].log_data[39].minminute := 27, [176].log_data[39].maxminute := 1, [176].log_data[39].valid := 1, [176].log_data[40].min := 7.5503016, [176].log_data[40].max := 7.5838275, [176].log_data[40].total := 27250.193, [176].log_data[40].time := 3600.0, [176].log_data[40].minminute := 30, [176].log_data[40].maxminute := 32, [176].log_data[40].valid := 1, [176].log_data[41].min := 0.09438281, [176].log_data[41].max := 0.12107837, [176].log_data[41].total := 379.78085, [176].log_data[41].time := 3600.0, [176].log_data[41].minminute := 1, [176].log_data[41].maxminute := 44, [176].log_data[41].valid := 1, [176].log_data[42].min := 2.2928205, [176].log_data[42].max := 2.2978847, [176].log_data[42].total := 8264.428, [176].log_data[42].time := 3600.0, [176].log_data[42].minminute := 54, [176].log_data[42].maxminute := 22, [176].log_data[42].valid := 1, [176].log_data[43].min := -0.27999878, [176].log_data[43].max := -0.26000214, [176].log_data[43].total := -969.35944, [176].log_data[43].time := 3600.0, [176].log_data[43].valid := 1, [176].log_data[44].min := -0.30000305, [176].log_data[44].max := -0.27999878, [176].log_data[44].total := -1080.0612, [176].log_data[44].time := 3600.0, [176].log_data[44].valid := 1, [176].log_data[45].time := 3600.0, [176].log_data[45].valid := 1, [176].log_data[46].time := 3600.0, [176].log_data[46].valid := 1, [176].log_data[47].time := 3600.0, [176].log_data[47].valid := 1, [176].log_data[48].min := 6.6725645, [176].log_data[48].max := 6.8014503, [176].log_data[48].total := 24349.217, [176].log_data[48].time := 3600.0, [176].log_data[48].maxminute := 8, [176].log_data[48].valid := 1, [176].log_data[49].min := 7.64159, [176].log_data[49].max := 9.454537, [176].log_data[49].total := 32845.09, [176].log_data[49].time := 3600.0, [176].log_data[49].maxminute := 55, [176].log_data[49].valid := 1, [176].log_data[50].min := 1.9997966, [176].log_data[50].max := 2.112625, [176].log_data[50].total := 7394.6826, [176].log_data[50].time := 3600.0,
        [176].log_data[50].minminute := 46, [176].log_data[50].maxminute := 59, [176].log_data[50].valid := 1, [176].log_data[51].time := 3600.0, [176].log_data[51].valid := 1, [176].log_data[52].min := -2.840004, [176].log_data[52].max := 0.11999512, [176].log_data[52].total := -6727.6313, [176].log_data[52].time := 3600.0, [176].log_data[52].minminute := 43, [176].log_data[52].valid := 1, [176].log_data[53].min := -2.4800034, [176].log_data[53].max := 0.22000122, [176].log_data[53].total := -6248.7065, [176].log_data[53].time := 3600.0, [176].log_data[53].minminute := 16, [176].log_data[53].maxminute := 25, [176].log_data[53].valid := 1, [176].log_data[54].max := 0.533, [176].log_data[54].total := 935.2089, [176].log_data[54].time := 3600.0, [176].log_data[54].maxminute := 43, [176].log_data[54].valid := 1, [176].log_data[55].max := 0.5205, [176].log_data[55].total := 939.1685, [176].log_data[55].time := 3600.0, [176].log_data[55].minminute := 3, [176].log_data[55].maxminute := 15, [176].log_data[55].valid := 1, [176].log_data[56].min := 0.16067745, [176].log_data[56].max := 0.16107002, [176].log_data[56].total := 578.9916, [176].log_data[56].time := 3600.0, [176].log_data[56].minminute := 19, [176].log_data[56].maxminute := 12, [176].log_data[56].valid := 1, [176].log_data[57].min := 0.34283584, [176].log_data[57].max := 0.34334624, [176].log_data[57].total := 1235.0238, [176].log_data[57].time := 3600.0, [176].log_data[57].minminute := 44, [176].log_data[57].valid := 1, [176].log_data[58].time := 3600.0, [176].log_data[58].valid := 1, [176].log_data[59].time := 3600.0, [176].log_data[59].valid := 1, [176].log_data[60].valid := 1, [176].log_data[61].valid := 1, [176].log_data[62].valid := 1, [176].log_data[63].valid := 1, [176].log_data[64].valid := 1, [176].log_data[65].valid := 1, [176].log_data[66].valid := 1, [176].log_data[67].valid := 1, [176].log_data[68].valid := 1, [176].log_data[69].valid := 1, [176].log_data[70].valid := 1, [176].log_data[71].valid := 1, [176].log_data[72].valid := 1, [176].log_data[73].valid := 1,
        [176].log_data[74].valid := 1, [176].log_data[75].valid := 1, [176].log_data[76].valid := 1, [176].log_data[77].valid := 1, [176].log_data[78].valid := 1, [176].log_data[79].valid := 1, [176].log_data[80].valid := 1, [176].log_data[81].valid := 1, [176].log_data[82].valid := 1, [176].log_data[83].valid := 1, [176].log_data[84].valid := 1, [176].log_data[85].valid := 1, [176].log_data[86].valid := 1, [176].log_data[87].valid := 1, [176].log_data[88].valid := 1, [176].log_data[89].valid := 1, [176].log_data[90].valid := 1, [176].log_data[91].valid := 1, [176].log_data[92].valid := 1, [176].log_data[93].valid := 1, [176].log_data[94].valid := 1, [176].log_data[95].valid := 1, [176].log_data[96].valid := 1, [176].log_data[97].valid := 1, [176].log_data[98].valid := 1, [176].log_data[99].valid := 1, [176].log_data[100].valid := 1, [176].log_data[101].valid := 1, [176].log_data[102].valid := 1, [176].log_data[103].valid := 1, [176].log_data[104].valid := 1, [176].log_data[105].valid := 1, [176].log_data[106].valid := 1, [176].log_data[107].valid := 1, [176].log_data[108].valid := 1, [176].log_data[109].valid := 1, [176].log_data[110].valid := 1, [176].log_data[111].valid := 1, [176].log_data[112].valid := 1, [176].log_data[113].valid := 1, [176].log_data[114].valid := 1, [176].log_data[115].valid := 1, [176].log_data[116].valid := 1, [176].log_data[117].valid := 1, [176].log_data[118].valid := 1, [176].log_data[119].valid := 1, [176].log_data[120].valid := 1, [176].log_data[121].valid := 1, [176].log_data[122].valid := 1, [176].log_data[123].valid := 1, [176].log_data[124].valid := 1, [176].time.Year := 2023, [176].time.Month := 1, [176].time.Day := 12, [176].time.Hour := 3, [176].time.Minute := 59, [176].time.Second := 59, [177].log_data[0].min := 1.0, [177].log_data[0].max := 1.0, [177].log_data[0].total := 3600.0,
        [177].log_data[0].time := 3600.0, [177].log_data[0].valid := 1, [177].log_data[1].time := 3600.0, [177].log_data[1].valid := 1, [177].log_data[2].time := 3600.0, [177].log_data[2].valid := 1, [177].log_data[3].time := 3600.0, [177].log_data[3].valid := 1, [177].log_data[4].time := 3600.0, [177].log_data[4].valid := 1, [177].log_data[5].time := 3600.0, [177].log_data[5].valid := 1, [177].log_data[6].time := 3600.0, [177].log_data[6].valid := 1, [177].log_data[7].time := 3600.0, [177].log_data[7].valid := 1, [177].log_data[8].time := 3600.0, [177].log_data[8].valid := 1, [177].log_data[9].time := 3600.0, [177].log_data[9].valid := 1, [177].log_data[10].min := 1.0, [177].log_data[10].max := 1.0, [177].log_data[10].total := 3600.0, [177].log_data[10].time := 3600.0, [177].log_data[10].valid := 1, [177].log_data[11].time := 3600.0, [177].log_data[11].valid := 1, [177].log_data[12].min := 1.0, [177].log_data[12].max := 1.0, [177].log_data[12].total := 3600.0, [177].log_data[12].time := 3600.0, [177].log_data[12].valid := 1, [177].log_data[13].min := 1.0, [177].log_data[13].max := 1.0, [177].log_data[13].total := 3600.0, [177].log_data[13].time := 3600.0, [177].log_data[13].valid := 1, [177].log_data[14].time := 3600.0, [177].log_data[14].valid := 1, [177].log_data[15].time := 3600.0, [177].log_data[15].valid := 1, [177].log_data[16].time := 3600.0, [177].log_data[16].valid := 1, [177].log_data[17].min := 1.0, [177].log_data[17].max := 1.0, [177].log_data[17].total := 3600.0, [177].log_data[17].time := 3600.0, [177].log_data[17].valid := 1, [177].log_data[18].time := 3600.0, [177].log_data[18].valid := 1, [177].log_data[19].time := 3600.0, [177].log_data[19].valid := 1, [177].log_data[20].time := 3600.0, [177].log_data[20].valid := 1, [177].log_data[21].min := 1.0, [177].log_data[21].max := 1.0, [177].log_data[21].total := 3600.0, [177].log_data[21].time := 3600.0, [177].log_data[21].valid := 1, [177].log_data[22].time := 3600.0,
        [177].log_data[22].valid := 1, [177].log_data[23].time := 3600.0, [177].log_data[23].valid := 1, [177].log_data[24].time := 3600.0, [177].log_data[24].valid := 1, [177].log_data[25].time := 3600.0, [177].log_data[25].valid := 1, [177].log_data[26].time := 3600.0, [177].log_data[26].valid := 1, [177].log_data[27].time := 3600.0, [177].log_data[27].valid := 1, [177].log_data[28].time := 3600.0, [177].log_data[28].valid := 1, [177].log_data[29].min := 1.0, [177].log_data[29].max := 1.0, [177].log_data[29].total := 3600.0, [177].log_data[29].time := 3600.0, [177].log_data[29].valid := 1, [177].log_data[30].min := 1.0, [177].log_data[30].max := 1.0, [177].log_data[30].total := 3600.0, [177].log_data[30].time := 3600.0, [177].log_data[30].valid := 1, [177].log_data[31].time := 3600.0, [177].log_data[31].valid := 1, [177].log_data[32].time := 3600.0, [177].log_data[32].valid := 1, [177].log_data[33].time := 3600.0, [177].log_data[33].valid := 1, [177].log_data[34].time := 3600.0, [177].log_data[34].valid := 1, [177].log_data[35].time := 3600.0, [177].log_data[35].valid := 1, [177].log_data[36].time := 3600.0, [177].log_data[36].valid := 1, [177].log_data[37].time := 3600.0, [177].log_data[37].valid := 1, [177].log_data[38].time := 3600.0, [177].log_data[38].valid := 1, [177].log_data[39].min := 0.9934107, [177].log_data[39].max := 1.0042459, [177].log_data[39].total := 3599.8289, [177].log_data[39].time := 3600.0, [177].log_data[39].minminute := 38, [177].log_data[39].maxminute := 9, [177].log_data[39].valid := 1, [177].log_data[40].min := 7.54453, [177].log_data[40].max := 7.586301, [177].log_data[40].total := 27250.268, [177].log_data[40].time := 3600.0, [177].log_data[40].minminute := 20, [177].log_data[40].maxminute := 22, [177].log_data[40].valid := 1, [177].log_data[41].min := 0.06965014, [177].log_data[41].max := 0.12107837, [177].log_data[41].total := 362.60077, [177].log_data[41].time := 3600.0, [177].log_data[41].minminute := 59, [177].log_data[41].maxminute := 6, [177].log_data[41].valid := 1,
        [177].log_data[42].min := 2.2929382, [177].log_data[42].max := 2.2980025, [177].log_data[42].total := 8264.365, [177].log_data[42].time := 3600.0, [177].log_data[42].minminute := 16, [177].log_data[42].maxminute := 47, [177].log_data[42].valid := 1, [177].log_data[43].min := -0.27999878, [177].log_data[43].max := -0.26000214, [177].log_data[43].total := -951.35785, [177].log_data[43].time := 3600.0, [177].log_data[43].valid := 1, [177].log_data[44].min := -0.30000305, [177].log_data[44].max := -0.27999878, [177].log_data[44].total := -1079.9807, [177].log_data[44].time := 3600.0, [177].log_data[44].maxminute := 9, [177].log_data[44].valid := 1, [177].log_data[45].time := 3600.0, [177].log_data[45].valid := 1, [177].log_data[46].time := 3600.0, [177].log_data[46].valid := 1, [177].log_data[47].time := 3600.0, [177].log_data[47].valid := 1, [177].log_data[48].min := 6.7522593, [177].log_data[48].max := 6.767099, [177].log_data[48].total := 24334.348, [177].log_data[48].time := 3600.0, [177].log_data[48].maxminute := 53, [177].log_data[48].valid := 1, [177].log_data[49].min := 9.412531, [177].log_data[49].max := 9.469455, [177].log_data[49].total := 33985.37, [177].log_data[49].time := 3600.0, [177].log_data[49].minminute := 6, [177].log_data[49].maxminute := 44, [177].log_data[49].valid := 1, [177].log_data[50].min := 2.1081495, [177].log_data[50].max := 2.119338, [177].log_data[50].total := 7612.295, [177].log_data[50].time := 3600.0, [177].log_data[50].minminute := 4, [177].log_data[50].maxminute := 42, [177].log_data[50].valid := 1, [177].log_data[51].time := 3600.0, [177].log_data[51].valid := 1, [177].log_data[52].min := -1.6200027, [177].log_data[52].max := -1.4000015, [177].log_data[52].total := -5412.9, [177].log_data[52].time := 3600.0, [177].log_data[52].minminute := 55, [177].log_data[52].valid := 1, [177].log_data[53].min := -1.4800034, [177].log_data[53].max := -1.2200012, [177].log_data[53].total := -4928.3027, [177].log_data[53].time := 3600.0, [177].log_data[53].minminute := 48, [177].log_data[53].valid := 1, [177].log_data[54].time := 3600.0, [177].log_data[54].valid := 1,
        [177].log_data[55].time := 3600.0, [177].log_data[55].valid := 1, [177].log_data[56].min := 0.16067745, [177].log_data[56].max := 0.16107002, [177].log_data[56].total := 578.9852, [177].log_data[56].time := 3600.0, [177].log_data[56].minminute := 26, [177].log_data[56].maxminute := 10, [177].log_data[56].valid := 1, [177].log_data[57].min := 0.3428751, [177].log_data[57].max := 0.34334624, [177].log_data[57].total := 1235.2053, [177].log_data[57].time := 3600.0, [177].log_data[57].minminute := 6, [177].log_data[57].maxminute := 34, [177].log_data[57].valid := 1, [177].log_data[58].time := 3600.0, [177].log_data[58].valid := 1, [177].log_data[59].time := 3600.0, [177].log_data[59].valid := 1, [177].log_data[60].valid := 1, [177].log_data[61].valid := 1, [177].log_data[62].valid := 1, [177].log_data[63].valid := 1, [177].log_data[64].valid := 1, [177].log_data[65].valid := 1, [177].log_data[66].valid := 1, [177].log_data[67].valid := 1, [177].log_data[68].valid := 1, [177].log_data[69].valid := 1, [177].log_data[70].valid := 1, [177].log_data[71].valid := 1, [177].log_data[72].valid := 1, [177].log_data[73].valid := 1, [177].log_data[74].valid := 1, [177].log_data[75].valid := 1, [177].log_data[76].valid := 1, [177].log_data[77].valid := 1, [177].log_data[78].valid := 1, [177].log_data[79].valid := 1, [177].log_data[80].valid := 1, [177].log_data[81].valid := 1, [177].log_data[82].valid := 1, [177].log_data[83].valid := 1, [177].log_data[84].valid := 1, [177].log_data[85].valid := 1, [177].log_data[86].valid := 1, [177].log_data[87].valid := 1, [177].log_data[88].valid := 1, [177].log_data[89].valid := 1, [177].log_data[90].valid := 1, [177].log_data[91].valid := 1, [177].log_data[92].valid := 1, [177].log_data[93].valid := 1, [177].log_data[94].valid := 1, [177].log_data[95].valid := 1, [177].log_data[96].valid := 1, [177].log_data[97].valid := 1, [177].log_data[98].valid := 1, [177].log_data[99].valid := 1,
        [177].log_data[100].valid := 1, [177].log_data[101].valid := 1, [177].log_data[102].valid := 1, [177].log_data[103].valid := 1, [177].log_data[104].valid := 1, [177].log_data[105].valid := 1, [177].log_data[106].valid := 1, [177].log_data[107].valid := 1, [177].log_data[108].valid := 1, [177].log_data[109].valid := 1, [177].log_data[110].valid := 1, [177].log_data[111].valid := 1, [177].log_data[112].valid := 1, [177].log_data[113].valid := 1, [177].log_data[114].valid := 1, [177].log_data[115].valid := 1, [177].log_data[116].valid := 1, [177].log_data[117].valid := 1, [177].log_data[118].valid := 1, [177].log_data[119].valid := 1, [177].log_data[120].valid := 1, [177].log_data[121].valid := 1, [177].log_data[122].valid := 1, [177].log_data[123].valid := 1, [177].log_data[124].valid := 1, [177].time.Year := 2023, [177].time.Month := 1, [177].time.Day := 12, [177].time.Hour := 4, [177].time.Minute := 59, [177].time.Second := 59, [178].log_data[0].min := 1.0, [178].log_data[0].max := 1.0, [178].log_data[0].total := 3600.0, [178].log_data[0].time := 3600.0, [178].log_data[0].valid := 1, [178].log_data[1].time := 3600.0, [178].log_data[1].valid := 1, [178].log_data[2].time := 3600.0, [178].log_data[2].valid := 1, [178].log_data[3].time := 3600.0, [178].log_data[3].valid := 1, [178].log_data[4].time := 3600.0, [178].log_data[4].valid := 1, [178].log_data[5].time := 3600.0, [178].log_data[5].valid := 1, [178].log_data[6].time := 3600.0, [178].log_data[6].valid := 1, [178].log_data[7].time := 3600.0, [178].log_data[7].valid := 1, [178].log_data[8].time := 3600.0, [178].log_data[8].valid := 1, [178].log_data[9].time := 3600.0, [178].log_data[9].valid := 1, [178].log_data[10].min := 1.0, [178].log_data[10].max := 1.0, [178].log_data[10].total := 3600.0, [178].log_data[10].time := 3600.0, [178].log_data[10].valid := 1, [178].log_data[11].time := 3600.0,
        [178].log_data[11].valid := 1, [178].log_data[12].min := 1.0, [178].log_data[12].max := 1.0, [178].log_data[12].total := 3600.0, [178].log_data[12].time := 3600.0, [178].log_data[12].valid := 1, [178].log_data[13].min := 1.0, [178].log_data[13].max := 1.0, [178].log_data[13].total := 3600.0, [178].log_data[13].time := 3600.0, [178].log_data[13].valid := 1, [178].log_data[14].time := 3600.0, [178].log_data[14].valid := 1, [178].log_data[15].time := 3600.0, [178].log_data[15].valid := 1, [178].log_data[16].time := 3600.0, [178].log_data[16].valid := 1, [178].log_data[17].min := 1.0, [178].log_data[17].max := 1.0, [178].log_data[17].total := 3600.0, [178].log_data[17].time := 3600.0, [178].log_data[17].valid := 1, [178].log_data[18].time := 3600.0, [178].log_data[18].valid := 1, [178].log_data[19].time := 3600.0, [178].log_data[19].valid := 1, [178].log_data[20].time := 3600.0, [178].log_data[20].valid := 1, [178].log_data[21].min := 1.0, [178].log_data[21].max := 1.0, [178].log_data[21].total := 3600.0, [178].log_data[21].time := 3600.0, [178].log_data[21].valid := 1, [178].log_data[22].time := 3600.0, [178].log_data[22].valid := 1, [178].log_data[23].time := 3600.0, [178].log_data[23].valid := 1, [178].log_data[24].time := 3600.0, [178].log_data[24].valid := 1, [178].log_data[25].time := 3600.0, [178].log_data[25].valid := 1, [178].log_data[26].time := 3600.0, [178].log_data[26].valid := 1, [178].log_data[27].time := 3600.0, [178].log_data[27].valid := 1, [178].log_data[28].time := 3600.0, [178].log_data[28].valid := 1, [178].log_data[29].min := 1.0, [178].log_data[29].max := 1.0, [178].log_data[29].total := 3600.0, [178].log_data[29].time := 3600.0, [178].log_data[29].valid := 1, [178].log_data[30].min := 1.0, [178].log_data[30].max := 1.0, [178].log_data[30].total := 3600.0, [178].log_data[30].time := 3600.0, [178].log_data[30].valid := 1, [178].log_data[31].time := 3600.0, [178].log_data[31].valid := 1, [178].log_data[32].time := 3600.0,
        [178].log_data[32].valid := 1, [178].log_data[33].time := 3600.0, [178].log_data[33].valid := 1, [178].log_data[34].time := 3600.0, [178].log_data[34].valid := 1, [178].log_data[35].time := 3600.0, [178].log_data[35].valid := 1, [178].log_data[36].time := 3600.0, [178].log_data[36].valid := 1, [178].log_data[37].time := 3600.0, [178].log_data[37].valid := 1, [178].log_data[38].time := 3600.0, [178].log_data[38].valid := 1, [178].log_data[39].min := 0.9947063, [178].log_data[39].max := 1.0041281, [178].log_data[39].total := 3599.6274, [178].log_data[39].time := 3600.0, [178].log_data[39].minminute := 4, [178].log_data[39].maxminute := 23, [178].log_data[39].valid := 1, [178].log_data[40].min := 7.548927, [178].log_data[40].max := 7.5934467, [178].log_data[40].total := 27243.66, [178].log_data[40].time := 3600.0, [178].log_data[40].minminute := 53, [178].log_data[40].maxminute := 49, [178].log_data[40].valid := 1, [178].log_data[41].min := 0.06572412, [178].log_data[41].max := 0.10458984, [178].log_data[41].total := 312.70587, [178].log_data[41].time := 3600.0, [178].log_data[41].minminute := 4, [178].log_data[41].maxminute := 35, [178].log_data[41].valid := 1, [178].log_data[42].min := 2.2927027, [178].log_data[42].max := 2.2976491, [178].log_data[42].total := 8264.086, [178].log_data[42].time := 3600.0, [178].log_data[42].minminute := 11, [178].log_data[42].maxminute := 5, [178].log_data[42].valid := 1, [178].log_data[43].min := -0.27999878, [178].log_data[43].max := -0.26000214, [178].log_data[43].total := -939.83484, [178].log_data[43].time := 3600.0, [178].log_data[43].valid := 1, [178].log_data[44].min := -0.30000305, [178].log_data[44].max := -0.27999878, [178].log_data[44].total := -1077.1659, [178].log_data[44].time := 3600.0, [178].log_data[44].maxminute := 3, [178].log_data[44].valid := 1, [178].log_data[45].time := 3600.0, [178].log_data[45].valid := 1, [178].log_data[46].time := 3600.0, [178].log_data[46].valid := 1, [178].log_data[47].time := 3600.0, [178].log_data[47].valid := 1, [178].log_data[48].min := 6.7635264, [178].log_data[48].max := 6.7739687,
        [178].log_data[48].total := 24367.092, [178].log_data[48].time := 3600.0, [178].log_data[48].maxminute := 59, [178].log_data[48].valid := 1, [178].log_data[49].min := 9.437656, [178].log_data[49].max := 9.497918, [178].log_data[49].total := 34080.44, [178].log_data[49].time := 3600.0, [178].log_data[49].minminute := 3, [178].log_data[49].maxminute := 57, [178].log_data[49].valid := 1, [178].log_data[50].min := 2.1093273, [178].log_data[50].max := 2.1189847, [178].log_data[50].total := 7613.2637, [178].log_data[50].time := 3600.0, [178].log_data[50].minminute := 57, [178].log_data[50].maxminute := 47, [178].log_data[50].valid := 1, [178].log_data[51].time := 3600.0, [178].log_data[51].valid := 1, [178].log_data[52].min := -1.6399994, [178].log_data[52].max := -1.4400024, [178].log_data[52].total := -5559.357, [178].log_data[52].time := 3600.0, [178].log_data[52].minminute := 30, [178].log_data[52].maxminute := 23, [178].log_data[52].valid := 1, [178].log_data[53].min := -1.5200043, [178].log_data[53].max := -1.340004, [178].log_data[53].total := -5169.0225, [178].log_data[53].time := 3600.0, [178].log_data[53].minminute := 44, [178].log_data[53].maxminute := 2, [178].log_data[53].valid := 1, [178].log_data[54].time := 3600.0, [178].log_data[54].valid := 1, [178].log_data[55].time := 3600.0, [178].log_data[55].valid := 1, [178].log_data[56].min := 0.16055967, [178].log_data[56].max := 0.16107002, [178].log_data[56].total := 578.83527, [178].log_data[56].time := 3600.0, [178].log_data[56].minminute := 36, [178].log_data[56].maxminute := 39, [178].log_data[56].valid := 1, [178].log_data[57].min := 0.34303212, [178].log_data[57].max := 0.34346402, [178].log_data[57].total := 1235.4823, [178].log_data[57].time := 3600.0, [178].log_data[57].maxminute := 57, [178].log_data[57].valid := 1, [178].log_data[58].time := 3600.0, [178].log_data[58].valid := 1, [178].log_data[59].time := 3600.0, [178].log_data[59].valid := 1, [178].log_data[60].valid := 1, [178].log_data[61].valid := 1, [178].log_data[62].valid := 1, [178].log_data[63].valid := 1, [178].log_data[64].valid := 1,
        [178].log_data[65].valid := 1, [178].log_data[66].valid := 1, [178].log_data[67].valid := 1, [178].log_data[68].valid := 1, [178].log_data[69].valid := 1, [178].log_data[70].valid := 1, [178].log_data[71].valid := 1, [178].log_data[72].valid := 1, [178].log_data[73].valid := 1, [178].log_data[74].valid := 1, [178].log_data[75].valid := 1, [178].log_data[76].valid := 1, [178].log_data[77].valid := 1, [178].log_data[78].valid := 1, [178].log_data[79].valid := 1, [178].log_data[80].valid := 1, [178].log_data[81].valid := 1, [178].log_data[82].valid := 1, [178].log_data[83].valid := 1, [178].log_data[84].valid := 1, [178].log_data[85].valid := 1, [178].log_data[86].valid := 1, [178].log_data[87].valid := 1, [178].log_data[88].valid := 1, [178].log_data[89].valid := 1, [178].log_data[90].valid := 1, [178].log_data[91].valid := 1, [178].log_data[92].valid := 1, [178].log_data[93].valid := 1, [178].log_data[94].valid := 1, [178].log_data[95].valid := 1, [178].log_data[96].valid := 1, [178].log_data[97].valid := 1, [178].log_data[98].valid := 1, [178].log_data[99].valid := 1, [178].log_data[100].valid := 1, [178].log_data[101].valid := 1, [178].log_data[102].valid := 1, [178].log_data[103].valid := 1, [178].log_data[104].valid := 1, [178].log_data[105].valid := 1, [178].log_data[106].valid := 1, [178].log_data[107].valid := 1, [178].log_data[108].valid := 1, [178].log_data[109].valid := 1, [178].log_data[110].valid := 1, [178].log_data[111].valid := 1, [178].log_data[112].valid := 1, [178].log_data[113].valid := 1, [178].log_data[114].valid := 1, [178].log_data[115].valid := 1, [178].log_data[116].valid := 1, [178].log_data[117].valid := 1, [178].log_data[118].valid := 1, [178].log_data[119].valid := 1, [178].log_data[120].valid := 1, [178].log_data[121].valid := 1, [178].log_data[122].valid := 1, [178].log_data[123].valid := 1, [178].log_data[124].valid := 1,
        [178].time.Year := 2023, [178].time.Month := 1, [178].time.Day := 12, [178].time.Hour := 5, [178].time.Minute := 59, [178].time.Second := 59, [179].log_data[0].min := 1.0, [179].log_data[0].max := 1.0, [179].log_data[0].total := 3600.0, [179].log_data[0].time := 3600.0, [179].log_data[0].valid := 1, [179].log_data[1].max := 1.0, [179].log_data[1].total := 563.0, [179].log_data[1].time := 3600.0, [179].log_data[1].maxminute := 39, [179].log_data[1].valid := 1, [179].log_data[2].max := 1.0, [179].log_data[2].total := 559.5, [179].log_data[2].time := 3600.0, [179].log_data[2].maxminute := 39, [179].log_data[2].valid := 1, [179].log_data[3].time := 3600.0, [179].log_data[3].valid := 1, [179].log_data[4].time := 3600.0, [179].log_data[4].valid := 1, [179].log_data[5].max := 1.0, [179].log_data[5].total := 226.5, [179].log_data[5].time := 3600.0, [179].log_data[5].maxminute := 42, [179].log_data[5].valid := 1, [179].log_data[6].time := 3600.0, [179].log_data[6].valid := 1, [179].log_data[7].time := 3600.0, [179].log_data[7].valid := 1, [179].log_data[8].max := 1.0, [179].log_data[8].total := 990.749, [179].log_data[8].time := 3600.0, [179].log_data[8].maxminute := 43, [179].log_data[8].valid := 1, [179].log_data[9].max := 1.0, [179].log_data[9].total := 987.249, [179].log_data[9].time := 3600.0, [179].log_data[9].maxminute := 43, [179].log_data[9].valid := 1, [179].log_data[10].min := 1.0, [179].log_data[10].max := 1.0, [179].log_data[10].total := 3600.0, [179].log_data[10].time := 3600.0, [179].log_data[10].valid := 1, [179].log_data[11].time := 3600.0, [179].log_data[11].valid := 1, [179].log_data[12].min := 1.0, [179].log_data[12].max := 1.0, [179].log_data[12].total := 3600.0, [179].log_data[12].time := 3600.0, [179].log_data[12].valid := 1, [179].log_data[13].min := 1.0, [179].log_data[13].max := 1.0, [179].log_data[13].total := 3600.0, [179].log_data[13].time := 3600.0,
        [179].log_data[13].valid := 1, [179].log_data[14].time := 3600.0, [179].log_data[14].valid := 1, [179].log_data[15].time := 3600.0, [179].log_data[15].valid := 1, [179].log_data[16].time := 3600.0, [179].log_data[16].valid := 1, [179].log_data[17].min := 1.0, [179].log_data[17].max := 1.0, [179].log_data[17].total := 3600.0, [179].log_data[17].time := 3600.0, [179].log_data[17].valid := 1, [179].log_data[18].time := 3600.0, [179].log_data[18].valid := 1, [179].log_data[19].time := 3600.0, [179].log_data[19].valid := 1, [179].log_data[20].time := 3600.0, [179].log_data[20].valid := 1, [179].log_data[21].min := 1.0, [179].log_data[21].max := 1.0, [179].log_data[21].total := 3600.0, [179].log_data[21].time := 3600.0, [179].log_data[21].valid := 1, [179].log_data[22].time := 3600.0, [179].log_data[22].valid := 1, [179].log_data[23].time := 3600.0, [179].log_data[23].valid := 1, [179].log_data[24].time := 3600.0, [179].log_data[24].valid := 1, [179].log_data[25].time := 3600.0, [179].log_data[25].valid := 1, [179].log_data[26].time := 3600.0, [179].log_data[26].valid := 1, [179].log_data[27].time := 3600.0, [179].log_data[27].valid := 1, [179].log_data[28].time := 3600.0, [179].log_data[28].valid := 1, [179].log_data[29].min := 1.0, [179].log_data[29].max := 1.0, [179].log_data[29].total := 3600.0, [179].log_data[29].time := 3600.0, [179].log_data[29].valid := 1, [179].log_data[30].min := 1.0, [179].log_data[30].max := 1.0, [179].log_data[30].total := 3600.0, [179].log_data[30].time := 3600.0, [179].log_data[30].valid := 1, [179].log_data[31].max := 1.0, [179].log_data[31].total := 529.749, [179].log_data[31].time := 3600.0, [179].log_data[31].maxminute := 51, [179].log_data[31].valid := 1, [179].log_data[32].max := 1.0, [179].log_data[32].total := 365.749, [179].log_data[32].time := 3600.0, [179].log_data[32].maxminute := 43, [179].log_data[32].valid := 1, [179].log_data[33].time := 3600.0, [179].log_data[33].valid := 1, [179].log_data[34].time := 3600.0,
        [179].log_data[34].valid := 1, [179].log_data[35].max := 1.0, [179].log_data[35].total := 348.749, [179].log_data[35].time := 3600.0, [179].log_data[35].maxminute := 54, [179].log_data[35].valid := 1, [179].log_data[36].max := 1.0, [179].log_data[36].total := 543.249, [179].log_data[36].time := 3600.0, [179].log_data[36].maxminute := 43, [179].log_data[36].valid := 1, [179].log_data[37].max := 7.012247, [179].log_data[37].total := 3420.6562, [179].log_data[37].time := 3600.0, [179].log_data[37].maxminute := 41, [179].log_data[37].valid := 1, [179].log_data[38].time := 3600.0, [179].log_data[38].valid := 1, [179].log_data[39].min := 0.9950596, [179].log_data[39].max := 1.02203, [179].log_data[39].total := 3606.1797, [179].log_data[39].time := 3600.0, [179].log_data[39].minminute := 29, [179].log_data[39].maxminute := 42, [179].log_data[39].valid := 1, [179].log_data[40].min := 7.548927, [179].log_data[40].max := 7.590423, [179].log_data[40].total := 27246.258, [179].log_data[40].time := 3600.0, [179].log_data[40].minminute := 47, [179].log_data[40].maxminute := 10, [179].log_data[40].valid := 1, [179].log_data[41].min := 0.07180932, [179].log_data[41].max := 0.09536426, [179].log_data[41].total := 306.74982, [179].log_data[41].time := 3600.0, [179].log_data[41].minminute := 13, [179].log_data[41].maxminute := 57, [179].log_data[41].valid := 1, [179].log_data[42].min := 2.2929382, [179].log_data[42].max := 2.2978847, [179].log_data[42].total := 8263.91, [179].log_data[42].time := 3600.0, [179].log_data[42].minminute := 46, [179].log_data[42].maxminute := 59, [179].log_data[42].valid := 1, [179].log_data[43].min := -0.26000214, [179].log_data[43].max := -0.23999786, [179].log_data[43].total := -935.93317, [179].log_data[43].time := 3600.0, [179].log_data[43].maxminute := 48, [179].log_data[43].valid := 1, [179].log_data[44].min := -0.30000305, [179].log_data[44].max := -0.27999878, [179].log_data[44].total := -1017.20996, [179].log_data[44].time := 3600.0, [179].log_data[44].valid := 1, [179].log_data[45].time := 3600.0, [179].log_data[45].valid := 1, [179].log_data[46].time := 3600.0,
        [179].log_data[46].valid := 1, [179].log_data[47].time := 3600.0, [179].log_data[47].valid := 1, [179].log_data[48].min := 6.690977, [179].log_data[48].max := 6.980899, [179].log_data[48].total := 24428.424, [179].log_data[48].time := 3600.0, [179].log_data[48].minminute := 59, [179].log_data[48].maxminute := 49, [179].log_data[48].valid := 1, [179].log_data[49].min := 7.171669, [179].log_data[49].max := 9.516369, [179].log_data[49].total := 32900.242, [179].log_data[49].time := 3600.0, [179].log_data[49].minminute := 59, [179].log_data[49].maxminute := 30, [179].log_data[49].valid := 1, [179].log_data[50].min := 2.0597441, [179].log_data[50].max := 2.151137, [179].log_data[50].total := 7597.4478, [179].log_data[50].time := 3600.0, [179].log_data[50].minminute := 47, [179].log_data[50].maxminute := 43, [179].log_data[50].valid := 1, [179].log_data[51].time := 3600.0, [179].log_data[51].valid := 1, [179].log_data[52].min := -4.2599945, [179].log_data[52].max := 0.11999512, [179].log_data[52].total := -6264.198, [179].log_data[52].time := 3600.0, [179].log_data[52].minminute := 43, [179].log_data[52].maxminute := 49, [179].log_data[52].valid := 1, [179].log_data[53].min := -3.9399948, [179].log_data[53].max := 0.22000122, [179].log_data[53].total := -5878.9165, [179].log_data[53].time := 3600.0, [179].log_data[53].minminute := 43, [179].log_data[53].maxminute := 53, [179].log_data[53].valid := 1, [179].log_data[54].max := 0.534, [179].log_data[54].total := 354.33246, [179].log_data[54].time := 3600.0, [179].log_data[54].maxminute := 51, [179].log_data[54].valid := 1, [179].log_data[55].max := 0.49449998, [179].log_data[55].total := 352.69998, [179].log_data[55].time := 3600.0, [179].log_data[55].maxminute := 43, [179].log_data[55].valid := 1, [179].log_data[56].min := 0.16055967, [179].log_data[56].max := 0.16103075, [179].log_data[56].total := 578.6617, [179].log_data[56].time := 3600.0, [179].log_data[56].minminute := 36, [179].log_data[56].maxminute := 5, [179].log_data[56].valid := 1, [179].log_data[57].min := 0.34311065, [179].log_data[57].max := 0.3435818, [179].log_data[57].total := 1235.9417,
        [179].log_data[57].time := 3600.0, [179].log_data[57].maxminute := 42, [179].log_data[57].valid := 1, [179].log_data[58].time := 3600.0, [179].log_data[58].valid := 1, [179].log_data[59].time := 3600.0, [179].log_data[59].valid := 1, [179].log_data[60].valid := 1, [179].log_data[61].valid := 1, [179].log_data[62].valid := 1, [179].log_data[63].valid := 1, [179].log_data[64].valid := 1, [179].log_data[65].valid := 1, [179].log_data[66].valid := 1, [179].log_data[67].valid := 1, [179].log_data[68].valid := 1, [179].log_data[69].valid := 1, [179].log_data[70].valid := 1, [179].log_data[71].valid := 1, [179].log_data[72].valid := 1, [179].log_data[73].valid := 1, [179].log_data[74].valid := 1, [179].log_data[75].valid := 1, [179].log_data[76].valid := 1, [179].log_data[77].valid := 1, [179].log_data[78].valid := 1, [179].log_data[79].valid := 1, [179].log_data[80].valid := 1, [179].log_data[81].valid := 1, [179].log_data[82].valid := 1, [179].log_data[83].valid := 1, [179].log_data[84].valid := 1, [179].log_data[85].valid := 1, [179].log_data[86].valid := 1, [179].log_data[87].valid := 1, [179].log_data[88].valid := 1, [179].log_data[89].valid := 1, [179].log_data[90].valid := 1, [179].log_data[91].valid := 1, [179].log_data[92].valid := 1, [179].log_data[93].valid := 1, [179].log_data[94].valid := 1, [179].log_data[95].valid := 1, [179].log_data[96].valid := 1, [179].log_data[97].valid := 1, [179].log_data[98].valid := 1, [179].log_data[99].valid := 1, [179].log_data[100].valid := 1, [179].log_data[101].valid := 1, [179].log_data[102].valid := 1, [179].log_data[103].valid := 1, [179].log_data[104].valid := 1, [179].log_data[105].valid := 1, [179].log_data[106].valid := 1, [179].log_data[107].valid := 1, [179].log_data[108].valid := 1, [179].log_data[109].valid := 1, [179].log_data[110].valid := 1, [179].log_data[111].valid := 1, [179].log_data[112].valid := 1,
        [179].log_data[113].valid := 1, [179].log_data[114].valid := 1, [179].log_data[115].valid := 1, [179].log_data[116].valid := 1, [179].log_data[117].valid := 1, [179].log_data[118].valid := 1, [179].log_data[119].valid := 1, [179].log_data[120].valid := 1, [179].log_data[121].valid := 1, [179].log_data[122].valid := 1, [179].log_data[123].valid := 1, [179].log_data[124].valid := 1, [179].time.Year := 2023, [179].time.Month := 1, [179].time.Day := 12, [179].time.Hour := 6, [179].time.Minute := 59, [179].time.Second := 59, [180].log_data[0].min := 1.0, [180].log_data[0].max := 1.0, [180].log_data[0].total := 3600.0, [180].log_data[0].time := 3600.0, [180].log_data[0].valid := 1, [180].log_data[1].time := 3600.0, [180].log_data[1].valid := 1, [180].log_data[2].time := 3600.0, [180].log_data[2].valid := 1, [180].log_data[3].time := 3600.0, [180].log_data[3].valid := 1, [180].log_data[4].time := 3600.0, [180].log_data[4].valid := 1, [180].log_data[5].time := 3600.0, [180].log_data[5].valid := 1, [180].log_data[6].time := 3600.0, [180].log_data[6].valid := 1, [180].log_data[7].time := 3600.0, [180].log_data[7].valid := 1, [180].log_data[8].min := 1.0, [180].log_data[8].max := 1.0, [180].log_data[8].total := 3600.0, [180].log_data[8].time := 3600.0, [180].log_data[8].valid := 1, [180].log_data[9].min := 1.0, [180].log_data[9].max := 1.0, [180].log_data[9].total := 3600.0, [180].log_data[9].time := 3600.0, [180].log_data[9].valid := 1, [180].log_data[10].min := 1.0, [180].log_data[10].max := 1.0, [180].log_data[10].total := 3600.0, [180].log_data[10].time := 3600.0, [180].log_data[10].valid := 1, [180].log_data[11].time := 3600.0, [180].log_data[11].valid := 1, [180].log_data[12].min := 1.0, [180].log_data[12].max := 1.0, [180].log_data[12].total := 3600.0, [180].log_data[12].time := 3600.0, [180].log_data[12].valid := 1, [180].log_data[13].min := 1.0,
        [180].log_data[13].max := 1.0, [180].log_data[13].total := 3600.0, [180].log_data[13].time := 3600.0, [180].log_data[13].valid := 1, [180].log_data[14].time := 3600.0, [180].log_data[14].valid := 1, [180].log_data[15].time := 3600.0, [180].log_data[15].valid := 1, [180].log_data[16].time := 3600.0, [180].log_data[16].valid := 1, [180].log_data[17].min := 1.0, [180].log_data[17].max := 1.0, [180].log_data[17].total := 3600.0, [180].log_data[17].time := 3600.0, [180].log_data[17].valid := 1, [180].log_data[18].time := 3600.0, [180].log_data[18].valid := 1, [180].log_data[19].time := 3600.0, [180].log_data[19].valid := 1, [180].log_data[20].time := 3600.0, [180].log_data[20].valid := 1, [180].log_data[21].min := 1.0, [180].log_data[21].max := 1.0, [180].log_data[21].total := 3600.0, [180].log_data[21].time := 3600.0, [180].log_data[21].valid := 1, [180].log_data[22].time := 3600.0, [180].log_data[22].valid := 1, [180].log_data[23].time := 3600.0, [180].log_data[23].valid := 1, [180].log_data[24].time := 3600.0, [180].log_data[24].valid := 1, [180].log_data[25].time := 3600.0, [180].log_data[25].valid := 1, [180].log_data[26].time := 3600.0, [180].log_data[26].valid := 1, [180].log_data[27].time := 3600.0, [180].log_data[27].valid := 1, [180].log_data[28].time := 3600.0, [180].log_data[28].valid := 1, [180].log_data[29].min := 1.0, [180].log_data[29].max := 1.0, [180].log_data[29].total := 3600.0, [180].log_data[29].time := 3600.0, [180].log_data[29].valid := 1, [180].log_data[30].min := 1.0, [180].log_data[30].max := 1.0, [180].log_data[30].total := 3600.0, [180].log_data[30].time := 3600.0, [180].log_data[30].valid := 1, [180].log_data[31].max := 1.0, [180].log_data[31].total := 1440.7471, [180].log_data[31].time := 3600.0, [180].log_data[31].valid := 1, [180].log_data[32].max := 1.0, [180].log_data[32].total := 1629.998, [180].log_data[32].time := 3600.0, [180].log_data[32].maxminute := 1, [180].log_data[32].valid := 1, [180].log_data[33].time := 3600.0,
        [180].log_data[33].valid := 1, [180].log_data[34].time := 3600.0, [180].log_data[34].valid := 1, [180].log_data[35].max := 1.0, [180].log_data[35].total := 1440.249, [180].log_data[35].time := 3600.0, [180].log_data[35].minminute := 3, [180].log_data[35].valid := 1, [180].log_data[36].max := 1.0, [180].log_data[36].total := 1629.7471, [180].log_data[36].time := 3600.0, [180].log_data[36].maxminute := 4, [180].log_data[36].valid := 1, [180].log_data[37].time := 3600.0, [180].log_data[37].valid := 1, [180].log_data[38].time := 3600.0, [180].log_data[38].valid := 1, [180].log_data[39].min := 0.99435294, [180].log_data[39].max := 1.0050704, [180].log_data[39].total := 3602.3376, [180].log_data[39].time := 3600.0, [180].log_data[39].minminute := 52, [180].log_data[39].maxminute := 55, [180].log_data[39].valid := 1, [180].log_data[40].min := 7.550027, [180].log_data[40].max := 7.5849276, [180].log_data[40].total := 27251.162, [180].log_data[40].time := 3600.0, [180].log_data[40].minminute := 6, [180].log_data[40].maxminute := 23, [180].log_data[40].valid := 1, [180].log_data[41].min := 0.074753664, [180].log_data[41].max := 0.13305224, [180].log_data[41].total := 369.9304, [180].log_data[41].time := 3600.0, [180].log_data[41].minminute := 20, [180].log_data[41].maxminute := 37, [180].log_data[41].valid := 1, [180].log_data[42].min := 2.2921138, [180].log_data[42].max := 2.2976491, [180].log_data[42].total := 8263.817, [180].log_data[42].time := 3600.0, [180].log_data[42].minminute := 55, [180].log_data[42].maxminute := 17, [180].log_data[42].valid := 1, [180].log_data[43].min := -0.26000214, [180].log_data[43].max := -0.23999786, [180].log_data[43].total := -935.89813, [180].log_data[43].time := 3600.0, [180].log_data[43].valid := 1, [180].log_data[44].min := -0.30000305, [180].log_data[44].max := -0.27999878, [180].log_data[44].total := -1014.9839, [180].log_data[44].time := 3600.0, [180].log_data[44].valid := 1, [180].log_data[45].time := 3600.0, [180].log_data[45].valid := 1, [180].log_data[46].time := 3600.0, [180].log_data[46].valid := 1, [180].log_data[47].time := 3600.0,
        [180].log_data[47].valid := 1, [180].log_data[48].min := 6.5920463, [180].log_data[48].max := 6.8050227, [180].log_data[48].total := 24205.549, [180].log_data[48].time := 3600.0, [180].log_data[48].minminute := 12, [180].log_data[48].maxminute := 27, [180].log_data[48].valid := 1, [180].log_data[49].min := 6.963599, [180].log_data[49].max := 9.429805, [180].log_data[49].total := 30416.59, [180].log_data[49].time := 3600.0, [180].log_data[49].minminute := 3, [180].log_data[49].maxminute := 58, [180].log_data[49].valid := 1, [180].log_data[50].min := 1.9997966, [180].log_data[50].max := 2.0977855, [180].log_data[50].total := 7386.0576, [180].log_data[50].time := 3600.0, [180].log_data[50].minminute := 59, [180].log_data[50].valid := 1, [180].log_data[51].time := 3600.0, [180].log_data[51].valid := 1, [180].log_data[52].min := -2.880005, [180].log_data[52].max := 0.13999939, [180].log_data[52].total := -7425.4326, [180].log_data[52].time := 3600.0, [180].log_data[52].minminute := 12, [180].log_data[52].maxminute := 32, [180].log_data[52].valid := 1, [180].log_data[53].min := -2.4400024, [180].log_data[53].max := 0.22000122, [180].log_data[53].total := -6818.342, [180].log_data[53].time := 3600.0, [180].log_data[53].minminute := 41, [180].log_data[53].maxminute := 4, [180].log_data[53].valid := 1, [180].log_data[54].max := 0.5405, [180].log_data[54].total := 1217.5094, [180].log_data[54].time := 3600.0, [180].log_data[54].maxminute := 12, [180].log_data[54].valid := 1, [180].log_data[55].max := 0.5185, [180].log_data[55].total := 1217.0707, [180].log_data[55].time := 3600.0, [180].log_data[55].minminute := 3, [180].log_data[55].maxminute := 36, [180].log_data[55].valid := 1, [180].log_data[56].min := 0.16048115, [180].log_data[56].max := 0.16091299, [180].log_data[56].total := 578.3234, [180].log_data[56].time := 3600.0, [180].log_data[56].minminute := 13, [180].log_data[56].maxminute := 6, [180].log_data[56].valid := 1, [180].log_data[57].min := 0.3418544, [180].log_data[57].max := 0.34362105, [180].log_data[57].total := 1232.4092, [180].log_data[57].time := 3600.0, [180].log_data[57].minminute := 20,
        [180].log_data[57].maxminute := 8, [180].log_data[57].valid := 1, [180].log_data[58].time := 3600.0, [180].log_data[58].valid := 1, [180].log_data[59].time := 3600.0, [180].log_data[59].valid := 1, [180].log_data[60].valid := 1, [180].log_data[61].valid := 1, [180].log_data[62].valid := 1, [180].log_data[63].valid := 1, [180].log_data[64].valid := 1, [180].log_data[65].valid := 1, [180].log_data[66].valid := 1, [180].log_data[67].valid := 1, [180].log_data[68].valid := 1, [180].log_data[69].valid := 1, [180].log_data[70].valid := 1, [180].log_data[71].valid := 1, [180].log_data[72].valid := 1, [180].log_data[73].valid := 1, [180].log_data[74].valid := 1, [180].log_data[75].valid := 1, [180].log_data[76].valid := 1, [180].log_data[77].valid := 1, [180].log_data[78].valid := 1, [180].log_data[79].valid := 1, [180].log_data[80].valid := 1, [180].log_data[81].valid := 1, [180].log_data[82].valid := 1, [180].log_data[83].valid := 1, [180].log_data[84].valid := 1, [180].log_data[85].valid := 1, [180].log_data[86].valid := 1, [180].log_data[87].valid := 1, [180].log_data[88].valid := 1, [180].log_data[89].valid := 1, [180].log_data[90].valid := 1, [180].log_data[91].valid := 1, [180].log_data[92].valid := 1, [180].log_data[93].valid := 1, [180].log_data[94].valid := 1, [180].log_data[95].valid := 1, [180].log_data[96].valid := 1, [180].log_data[97].valid := 1, [180].log_data[98].valid := 1, [180].log_data[99].valid := 1, [180].log_data[100].valid := 1, [180].log_data[101].valid := 1, [180].log_data[102].valid := 1, [180].log_data[103].valid := 1, [180].log_data[104].valid := 1, [180].log_data[105].valid := 1, [180].log_data[106].valid := 1, [180].log_data[107].valid := 1, [180].log_data[108].valid := 1, [180].log_data[109].valid := 1, [180].log_data[110].valid := 1, [180].log_data[111].valid := 1, [180].log_data[112].valid := 1, [180].log_data[113].valid := 1,
        [180].log_data[114].valid := 1, [180].log_data[115].valid := 1, [180].log_data[116].valid := 1, [180].log_data[117].valid := 1, [180].log_data[118].valid := 1, [180].log_data[119].valid := 1, [180].log_data[120].valid := 1, [180].log_data[121].valid := 1, [180].log_data[122].valid := 1, [180].log_data[123].valid := 1, [180].log_data[124].valid := 1, [180].time.Year := 2023, [180].time.Month := 1, [180].time.Day := 12, [180].time.Hour := 7, [180].time.Minute := 59, [180].time.Second := 59, [181].log_data[0].min := 1.0, [181].log_data[0].max := 1.0, [181].log_data[0].total := 3600.0, [181].log_data[0].time := 3600.0, [181].log_data[0].valid := 1, [181].log_data[1].max := 1.0, [181].log_data[1].total := 90.249, [181].log_data[1].time := 3600.0, [181].log_data[1].maxminute := 58, [181].log_data[1].valid := 1, [181].log_data[2].max := 1.0, [181].log_data[2].total := 86.749, [181].log_data[2].time := 3600.0, [181].log_data[2].maxminute := 58, [181].log_data[2].valid := 1, [181].log_data[3].time := 3600.0, [181].log_data[3].valid := 1, [181].log_data[4].time := 3600.0, [181].log_data[4].valid := 1, [181].log_data[5].time := 3600.0, [181].log_data[5].valid := 1, [181].log_data[6].time := 3600.0, [181].log_data[6].valid := 1, [181].log_data[7].time := 3600.0, [181].log_data[7].valid := 1, [181].log_data[8].max := 1.0, [181].log_data[8].total := 111.251, [181].log_data[8].time := 3600.0, [181].log_data[8].minminute := 1, [181].log_data[8].valid := 1, [181].log_data[9].max := 1.0, [181].log_data[9].total := 111.251, [181].log_data[9].time := 3600.0, [181].log_data[9].minminute := 1, [181].log_data[9].valid := 1, [181].log_data[10].min := 1.0, [181].log_data[10].max := 1.0, [181].log_data[10].total := 3600.0, [181].log_data[10].time := 3600.0, [181].log_data[10].valid := 1, [181].log_data[11].time := 3600.0, [181].log_data[11].valid := 1, [181].log_data[12].min := 1.0,
        [181].log_data[12].max := 1.0, [181].log_data[12].total := 3600.0, [181].log_data[12].time := 3600.0, [181].log_data[12].valid := 1, [181].log_data[13].min := 1.0, [181].log_data[13].max := 1.0, [181].log_data[13].total := 3600.0, [181].log_data[13].time := 3600.0, [181].log_data[13].valid := 1, [181].log_data[14].time := 3600.0, [181].log_data[14].valid := 1, [181].log_data[15].time := 3600.0, [181].log_data[15].valid := 1, [181].log_data[16].time := 3600.0, [181].log_data[16].valid := 1, [181].log_data[17].min := 1.0, [181].log_data[17].max := 1.0, [181].log_data[17].total := 3600.0, [181].log_data[17].time := 3600.0, [181].log_data[17].valid := 1, [181].log_data[18].time := 3600.0, [181].log_data[18].valid := 1, [181].log_data[19].time := 3600.0, [181].log_data[19].valid := 1, [181].log_data[20].time := 3600.0, [181].log_data[20].valid := 1, [181].log_data[21].min := 1.0, [181].log_data[21].max := 1.0, [181].log_data[21].total := 3600.0, [181].log_data[21].time := 3600.0, [181].log_data[21].valid := 1, [181].log_data[22].time := 3600.0, [181].log_data[22].valid := 1, [181].log_data[23].time := 3600.0, [181].log_data[23].valid := 1, [181].log_data[24].time := 3600.0, [181].log_data[24].valid := 1, [181].log_data[25].time := 3600.0, [181].log_data[25].valid := 1, [181].log_data[26].time := 3600.0, [181].log_data[26].valid := 1, [181].log_data[27].time := 3600.0, [181].log_data[27].valid := 1, [181].log_data[28].time := 3600.0, [181].log_data[28].valid := 1, [181].log_data[29].min := 1.0, [181].log_data[29].max := 1.0, [181].log_data[29].total := 3600.0, [181].log_data[29].time := 3600.0, [181].log_data[29].valid := 1, [181].log_data[30].min := 1.0, [181].log_data[30].max := 1.0, [181].log_data[30].total := 3600.0, [181].log_data[30].time := 3600.0, [181].log_data[30].valid := 1, [181].log_data[31].max := 1.0, [181].log_data[31].total := 115.0, [181].log_data[31].time := 3600.0, [181].log_data[31].minminute := 1, [181].log_data[31].valid := 1,
        [181].log_data[32].time := 3600.0, [181].log_data[32].valid := 1, [181].log_data[33].time := 3600.0, [181].log_data[33].valid := 1, [181].log_data[34].time := 3600.0, [181].log_data[34].valid := 1, [181].log_data[35].max := 1.0, [181].log_data[35].total := 115.251, [181].log_data[35].time := 3600.0, [181].log_data[35].minminute := 1, [181].log_data[35].valid := 1, [181].log_data[36].time := 3600.0, [181].log_data[36].valid := 1, [181].log_data[37].max := 7.5579367, [181].log_data[37].total := 662.0562, [181].log_data[37].time := 3600.0, [181].log_data[37].maxminute := 59, [181].log_data[37].valid := 1, [181].log_data[38].time := 3600.0, [181].log_data[38].valid := 1, [181].log_data[39].min := 0.994824, [181].log_data[39].max := 1.0111947, [181].log_data[39].total := 3602.426, [181].log_data[39].time := 3600.0, [181].log_data[39].minminute := 12, [181].log_data[39].maxminute := 59, [181].log_data[39].valid := 1, [181].log_data[40].min := 7.5588202, [181].log_data[40].max := 7.5777817, [181].log_data[40].total := 27257.479, [181].log_data[40].time := 3600.0, [181].log_data[40].minminute := 34, [181].log_data[40].maxminute := 2, [181].log_data[40].valid := 1, [181].log_data[41].min := 0.07671655, [181].log_data[41].max := 0.11793774, [181].log_data[41].total := 355.52765, [181].log_data[41].time := 3600.0, [181].log_data[41].minminute := 49, [181].log_data[41].maxminute := 19, [181].log_data[41].valid := 1, [181].log_data[42].min := 2.292467, [181].log_data[42].max := 2.297767, [181].log_data[42].total := 8263.808, [181].log_data[42].time := 3600.0, [181].log_data[42].minminute := 24, [181].log_data[42].maxminute := 24, [181].log_data[42].valid := 1, [181].log_data[43].min := -0.26000214, [181].log_data[43].max := -0.26000214, [181].log_data[43].total := -935.9732, [181].log_data[43].time := 3600.0, [181].log_data[43].valid := 1, [181].log_data[44].min := -0.30000305, [181].log_data[44].max := -0.27999878, [181].log_data[44].total := -1037.9419, [181].log_data[44].time := 3600.0, [181].log_data[44].valid := 1, [181].log_data[45].time := 3600.0, [181].log_data[45].valid := 1,
        [181].log_data[46].time := 3600.0, [181].log_data[46].valid := 1, [181].log_data[47].time := 3600.0, [181].log_data[47].valid := 1, [181].log_data[48].min := 6.74319, [181].log_data[48].max := 6.751435, [181].log_data[48].total := 24286.887, [181].log_data[48].time := 3600.0, [181].log_data[48].minminute := 7, [181].log_data[48].maxminute := 54, [181].log_data[48].valid := 1, [181].log_data[49].min := 9.414102, [181].log_data[49].max := 9.481822, [181].log_data[49].total := 34010.18, [181].log_data[49].time := 3600.0, [181].log_data[49].minminute := 4, [181].log_data[49].maxminute := 58, [181].log_data[49].valid := 1, [181].log_data[50].min := 1.9988544, [181].log_data[50].max := 2.1202803, [181].log_data[50].total := 7589.7373, [181].log_data[50].time := 3600.0, [181].log_data[50].minminute := 1, [181].log_data[50].maxminute := 48, [181].log_data[50].valid := 1, [181].log_data[51].time := 3600.0, [181].log_data[51].valid := 1, [181].log_data[52].min := -2.6200027, [181].log_data[52].max := 0.039993286, [181].log_data[52].total := -5288.511, [181].log_data[52].time := 3600.0, [181].log_data[52].maxminute := 2, [181].log_data[52].valid := 1, [181].log_data[53].min := -2.4400024, [181].log_data[53].max := -0.16000366, [181].log_data[53].total := -5004.0103, [181].log_data[53].time := 3600.0, [181].log_data[53].maxminute := 1, [181].log_data[53].valid := 1, [181].log_data[54].max := 0.4285, [181].log_data[54].total := 46.39152, [181].log_data[54].time := 3600.0, [181].log_data[54].minminute := 1, [181].log_data[54].valid := 1, [181].log_data[55].max := 0.4285, [181].log_data[55].total := 46.48322, [181].log_data[55].time := 3600.0, [181].log_data[55].minminute := 1, [181].log_data[55].maxminute := 1, [181].log_data[55].valid := 1, [181].log_data[56].min := 0.1605204, [181].log_data[56].max := 0.16091299, [181].log_data[56].total := 578.3399, [181].log_data[56].time := 3600.0, [181].log_data[56].minminute := 7, [181].log_data[56].maxminute := 48, [181].log_data[56].valid := 1, [181].log_data[57].min := 0.34189364, [181].log_data[57].max := 0.34224698, [181].log_data[57].total := 1231.2078,
        [181].log_data[57].time := 3600.0, [181].log_data[57].minminute := 2, [181].log_data[57].maxminute := 10, [181].log_data[57].valid := 1, [181].log_data[58].time := 3600.0, [181].log_data[58].valid := 1, [181].log_data[59].time := 3600.0, [181].log_data[59].valid := 1, [181].log_data[60].valid := 1, [181].log_data[61].valid := 1, [181].log_data[62].valid := 1, [181].log_data[63].valid := 1, [181].log_data[64].valid := 1, [181].log_data[65].valid := 1, [181].log_data[66].valid := 1, [181].log_data[67].valid := 1, [181].log_data[68].valid := 1, [181].log_data[69].valid := 1, [181].log_data[70].valid := 1, [181].log_data[71].valid := 1, [181].log_data[72].valid := 1, [181].log_data[73].valid := 1, [181].log_data[74].valid := 1, [181].log_data[75].valid := 1, [181].log_data[76].valid := 1, [181].log_data[77].valid := 1, [181].log_data[78].valid := 1, [181].log_data[79].valid := 1, [181].log_data[80].valid := 1, [181].log_data[81].valid := 1, [181].log_data[82].valid := 1, [181].log_data[83].valid := 1, [181].log_data[84].valid := 1, [181].log_data[85].valid := 1, [181].log_data[86].valid := 1, [181].log_data[87].valid := 1, [181].log_data[88].valid := 1, [181].log_data[89].valid := 1, [181].log_data[90].valid := 1, [181].log_data[91].valid := 1, [181].log_data[92].valid := 1, [181].log_data[93].valid := 1, [181].log_data[94].valid := 1, [181].log_data[95].valid := 1, [181].log_data[96].valid := 1, [181].log_data[97].valid := 1, [181].log_data[98].valid := 1, [181].log_data[99].valid := 1, [181].log_data[100].valid := 1, [181].log_data[101].valid := 1, [181].log_data[102].valid := 1, [181].log_data[103].valid := 1, [181].log_data[104].valid := 1, [181].log_data[105].valid := 1, [181].log_data[106].valid := 1, [181].log_data[107].valid := 1, [181].log_data[108].valid := 1, [181].log_data[109].valid := 1, [181].log_data[110].valid := 1, [181].log_data[111].valid := 1,
        [181].log_data[112].valid := 1, [181].log_data[113].valid := 1, [181].log_data[114].valid := 1, [181].log_data[115].valid := 1, [181].log_data[116].valid := 1, [181].log_data[117].valid := 1, [181].log_data[118].valid := 1, [181].log_data[119].valid := 1, [181].log_data[120].valid := 1, [181].log_data[121].valid := 1, [181].log_data[122].valid := 1, [181].log_data[123].valid := 1, [181].log_data[124].valid := 1, [181].time.Year := 2023, [181].time.Month := 1, [181].time.Day := 12, [181].time.Hour := 8, [181].time.Minute := 59, [181].time.Second := 59, [182].log_data[0].min := 1.0, [182].log_data[0].max := 1.0, [182].log_data[0].total := 3600.0, [182].log_data[0].time := 3600.0, [182].log_data[0].valid := 1, [182].log_data[1].max := 1.0, [182].log_data[1].total := 448.251, [182].log_data[1].time := 3600.0, [182].log_data[1].minminute := 7, [182].log_data[1].valid := 1, [182].log_data[2].max := 1.0, [182].log_data[2].total := 448.251, [182].log_data[2].time := 3600.0, [182].log_data[2].minminute := 7, [182].log_data[2].valid := 1, [182].log_data[3].time := 3600.0, [182].log_data[3].valid := 1, [182].log_data[4].time := 3600.0, [182].log_data[4].valid := 1, [182].log_data[5].max := 1.0, [182].log_data[5].total := 230.5, [182].log_data[5].time := 3600.0, [182].log_data[5].maxminute := 1, [182].log_data[5].valid := 1, [182].log_data[6].time := 3600.0, [182].log_data[6].valid := 1, [182].log_data[7].time := 3600.0, [182].log_data[7].valid := 1, [182].log_data[8].max := 1.0, [182].log_data[8].total := 3454.249, [182].log_data[8].time := 3600.0, [182].log_data[8].maxminute := 2, [182].log_data[8].valid := 1, [182].log_data[9].max := 1.0, [182].log_data[9].total := 3450.749, [182].log_data[9].time := 3600.0, [182].log_data[9].maxminute := 2, [182].log_data[9].valid := 1, [182].log_data[10].min := 1.0, [182].log_data[10].max := 1.0, [182].log_data[10].total := 3600.0,
        [182].log_data[10].time := 3600.0, [182].log_data[10].valid := 1, [182].log_data[11].time := 3600.0, [182].log_data[11].valid := 1, [182].log_data[12].min := 1.0, [182].log_data[12].max := 1.0, [182].log_data[12].total := 3600.0, [182].log_data[12].time := 3600.0, [182].log_data[12].valid := 1, [182].log_data[13].min := 1.0, [182].log_data[13].max := 1.0, [182].log_data[13].total := 3600.0, [182].log_data[13].time := 3600.0, [182].log_data[13].valid := 1, [182].log_data[14].time := 3600.0, [182].log_data[14].valid := 1, [182].log_data[15].time := 3600.0, [182].log_data[15].valid := 1, [182].log_data[16].time := 3600.0, [182].log_data[16].valid := 1, [182].log_data[17].min := 1.0, [182].log_data[17].max := 1.0, [182].log_data[17].total := 3600.0, [182].log_data[17].time := 3600.0, [182].log_data[17].valid := 1, [182].log_data[18].time := 3600.0, [182].log_data[18].valid := 1, [182].log_data[19].time := 3600.0, [182].log_data[19].valid := 1, [182].log_data[20].time := 3600.0, [182].log_data[20].valid := 1, [182].log_data[21].min := 1.0, [182].log_data[21].max := 1.0, [182].log_data[21].total := 3600.0, [182].log_data[21].time := 3600.0, [182].log_data[21].valid := 1, [182].log_data[22].time := 3600.0, [182].log_data[22].valid := 1, [182].log_data[23].time := 3600.0, [182].log_data[23].valid := 1, [182].log_data[24].time := 3600.0, [182].log_data[24].valid := 1, [182].log_data[25].time := 3600.0, [182].log_data[25].valid := 1, [182].log_data[26].time := 3600.0, [182].log_data[26].valid := 1, [182].log_data[27].time := 3600.0, [182].log_data[27].valid := 1, [182].log_data[28].time := 3600.0, [182].log_data[28].valid := 1, [182].log_data[29].min := 1.0, [182].log_data[29].max := 1.0, [182].log_data[29].total := 3600.0, [182].log_data[29].time := 3600.0, [182].log_data[29].valid := 1, [182].log_data[30].min := 1.0, [182].log_data[30].max := 1.0, [182].log_data[30].total := 3600.0, [182].log_data[30].time := 3600.0, [182].log_data[30].valid := 1,
